// TwinCAT 3 PLC project FactoryIOPLCProject
// ProgramVersion: 3.1.4026.24
// libraries:
//   Tc2_ModbusSrv, * (Beckhoff Automation GmbH)
//   Tc2_Standard, * (Beckhoff Automation GmbH)
//   Tc2_System, * (Beckhoff Automation GmbH)
//   Tc2_Utilities, * (Beckhoff Automation GmbH)
// project tree:
//   DUTs/Communication/ADS/ ADSCommunicationInterface.TcDUT (not stored)
//   DUTs/HMI/Header/ HMIHeader.TcDUT
//   DUTs/HMI/MachineSection/ HMIMovementForkInterface.TcDUT, HMIMovementInterface.TcDUT, HMIRFIDControlInterface.TcDUT (not stored), HMIRFIDDataInterface.TcDUT (not stored), HMIRFIDInterface.TcDUT, HMIRFIDStatusInterface.TcDUT, HMIRuncontrolInterface.TcDUT, HMIWindowSwitch.TcDUT, HMIWorkpieceInterface.TcDUT, MachineSection.TcDUT, MachineSectionHMIInterface.TcDUT
//   DUTs/HMI/NumericalInput/ HMIButtonNumericalInputInterface.TcDUT, HMINumericalInputInterface.TcDUT (not stored), HMINumericalInputLineInterface.TcDUT
//   DUTs/HMI/SettingLine/ HMIButtonSettingLineInterface.TcDUT, HMISettingLineInterface.TcDUT
//   DUTs/OperatingMode/ ActionState.TcDUT, FaultWarningState.TcDUT (not stored), HMIActionState.TcDUT, HMIInterfaceOperatingMode.TcDUT (not stored), HMIToPLCOperatingMode.TcDUT, OperatingMode.TcDUT (not stored), OperatingModeHomeing.TcDUT, PLCToHMIOperatingMode.TcDUT
//   DUTs/PickPlace/ PickPlacePosition.TcDUT
//   DUTs/PositingBar/ PositingBarAlignmentDirection.TcDUT (not stored)
//   DUTs/Program/PickPlace/ PickPlaceSteps.TcDUT
//   DUTs/Program/Warehouse/ StackerCraneSteps.TcDUT (not stored)
//   DUTs/RFID/ RFIDReadSerialnumberStates.TcDUT, RFIDReadWriteDataStates.TcDUT (not stored)
//   DUTs/VisionSensor/ VisionSensorParttype.TcDUT (not stored)
//   GVLs/ ADS_Communication.TcGVL, Elevator.TcGVL, Emitter.TcGVL, Foerderband.TcGVL, GVL.TcGVL, HMI.TcGVL, PickPlace.TcGVL, PositioningBar.TcGVL, Remover.TcGVL, RFID.TcGVL, VisionSensor.TcGVL, Warehouse.TcGVL, _OperatingMode.TcGVL, _IO.TcGVL
//   / PlcTask.TcTTO (not stored)
//   POUs/Programm/ADS/ Call_ADSCommunication.TcPOU
//   POUs/Programm/Aufzug/ Call_Aufzug.TcPOU
//   POUs/Programm/Emitter/ Call_Emitter.TcPOU
//   POUs/Programm/Foerderband/ Call_Foerderband.TcPOU
//   POUs/Programm/HMI/ Call_HMI.TcPOU
//   POUs/Programm/ MAIN.TcPOU, SignalmappingInput.TcPOU, SignalmappingOutput.TcPOU
//   POUs/Programm/OperatingMode/ Call_OperatingMode.TcPOU
//   POUs/Programm/PickPlace/ Call_PickPlace.TcPOU
//   POUs/Programm/PositingBar/ Call_PositingBar.TcPOU
//   POUs/Programm/Remover/ Call_Remover.TcPOU
//   POUs/Programm/RFID/ Call_RFID.TcPOU
//   POUs/Programm/VisionSensor/ Call_VisionSensor.TcPOU
//   POUs/Programm/Warehouse/ Call_Warehouse.TcPOU
//   POUs/Vorlagen/AnalogValueHandling/ FC_AnalogInputValueHandling.TcPOU, FC_AnalogOutputValueHandling.TcPOU (not stored)
//   POUs/Vorlagen/Aufzug/ FB_Elevator.TcPOU
//   POUs/Vorlagen/Communication/ADS/ FB_ADSCommunicationStatus.TcPOU
//   POUs/Vorlagen/Emitter/ FB_Emitter.TcPOU
//   POUs/Vorlagen/Foerderband/ FB_Foerderband.TcPOU
//   POUs/Vorlagen/HMI/ FB_HMIHeader.TcPOU, FC_InitializingSettingLines.TcPOU
//   POUs/Vorlagen/OperatingMode/ FB_OperatingMode.TcPOU
//   POUs/Vorlagen/PickPlace/ FB_PickPlace_DigitalAnalog.TcPOU
//   POUs/Vorlagen/PositingBar/ FB_PositingBar.TcPOU
//   POUs/Vorlagen/Remover/ FB_Remover.TcPOU
//   POUs/Vorlagen/RFID/ FB_RFID.TcPOU
//   POUs/Vorlagen/VisionSensor/ FB_VisionSensor.TcPOU
//   POUs/Vorlagen/Warehouse/ FB_StackerCrane_Analog.TcPOU (not stored), FB_StackerCrane_Numerical.TcPOU
// real-time tasks:
//   TASK PlcTask: cycle T#10ms, priority 20, ADS port 350

// ---- DUTs/HMI/Header/HMIHeader.TcDUT
TYPE HMIHeader :
STRUCT
	PathOperatingMode	:	STRING;
	PathMachineState	:	STRING;
	NameApplication	:	STRING;
	ErrorIsActive	:	BOOL;
	State	:	INT;
END_STRUCT
END_TYPE

// ---- DUTs/HMI/MachineSection/HMIMovementForkInterface.TcDUT
TYPE HMIMovementForkInterface :
STRUCT
	ForkMovementButtons	:	ARRAY [1..8] of HMIButtonMachineSection;
END_STRUCT
END_TYPE

// ---- DUTs/HMI/MachineSection/HMIMovementInterface.TcDUT
TYPE HMIMovementInterface :
STRUCT
	MovementSettingLines	:	ARRAY [1..3] of HMISettingLineInterface;
END_STRUCT
END_TYPE

// ---- DUTs/HMI/MachineSection/HMIRFIDInterface.TcDUT
TYPE HMIRFIDInterface :
STRUCT
	PermissionHardware	:	BOOL;
	PartPresent	:	BOOL;
	ExecuteCommand	:	BOOL;
	FMReading	:	BOOL;
	FMWritting	:	BOOL;
	ErrorActive	:	BOOL;
	SelectedCommand	:	WORD;
	ReadValue	:	WORD;
	WriteValue	:	WORD;
	SelectedMemoryIndex	:	WORD;
	StatusReader	:	WORD;
	CommandID	:	WORD;
	AllReadData	:	ARRAY[0..127] OF WORD;
	AllWriteData	:	ARRAY[0..127] OF WORD;
END_STRUCT
END_TYPE

// ---- DUTs/HMI/MachineSection/HMIRFIDStatusInterface.TcDUT
TYPE HMIRFIDStatusInterface :
STRUCT
	PermissionHardware	:	BOOL;
	PartPresent	:	BOOL;
	ErrorActive	:	BOOL;
	FMReading	:	BOOL;
	FMWritting	:	BOOL;
END_STRUCT
END_TYPE

// ---- DUTs/HMI/MachineSection/HMIRuncontrolInterface.TcDUT
TYPE HMIRuncontrolInterface :
STRUCT
	RuncontrolButtons	:	ARRAY [1..10] of HMIButtonMachineSection;
END_STRUCT
END_TYPE

// ---- DUTs/HMI/MachineSection/HMIWindowSwitch.TcDUT
TYPE HMIWindowSwitch :
STRUCT
	MinPage	:	INT;
	MaxPage	:	INT;
	SelectedPage	:	INT;
	SelectedTab	:	STRING;
	NextPageIsEnabled	:	BOOL;
	NextPageIsPressed	:	BOOL;
	PreviousPageIsEnabled	:	BOOL;
	PreviousPageIsPressed	:	BOOL;
END_STRUCT
END_TYPE

// ---- DUTs/HMI/MachineSection/HMIWorkpieceInterface.TcDUT
TYPE HMIWorkpieceInterface :
STRUCT
	WorkpieceSettingLines	:	ARRAY[1..3] of HMISettingLineInterface;	
END_STRUCT
END_TYPE

// ---- DUTs/HMI/MachineSection/MachineSection.TcDUT
{attribute 'qualified_only'}
{attribute 'strict'}
{attribute 'to_string'}
TYPE MachineSection :
(
	None := 0,
	Conveyor,
	Emitter,
	Elevator,
	StackerCrane,
	RFID,
	PositingBar,
	PickPlace,
	Remover
);
END_TYPE

// ---- DUTs/HMI/MachineSection/MachineSectionHMIInterface.TcDUT
TYPE MachineSectionHMIInterface :
STRUCT
	ActiveMachineSection : MachineSection;
	SelectedActor : INT;
	PageSwitch	:	HMIWindowSwitch;
	Movements : HMIMovementInterface;
	Forks : HMIMovementForkInterface;
	Runcontrols : HMIRuncontrolInterface;
	RFID : HMIRFIDInterface;
	Workpiece : HMIWorkpieceInterface;
END_STRUCT
END_TYPE

// ---- DUTs/HMI/NumericalInput/HMIButtonNumericalInputInterface.TcDUT
TYPE HMIButtonNumericalInputInterface :
STRUCT
	IsEnabled	:	BOOL;
	IsPressed	:	BOOL;
	InPosition	:	BOOL;
	IsVisibleButton	:	BOOL;
	CaptionButton	:	STRING;
	PathImageButton	:	STRING;
END_STRUCT
END_TYPE

// ---- DUTs/HMI/NumericalInput/HMINumericalInputLineInterface.TcDUT
TYPE HMINumericalInputLineInterface :
STRUCT
	CaptionDescription	:	STRING;
	UnitInput	:	STRING;
	ValueInput	:	REAL;
	IsEnabledInput	:	BOOL;
END_STRUCT
END_TYPE

// ---- DUTs/HMI/SettingLine/HMIButtonSettingLineInterface.TcDUT
TYPE HMIButtonSettingLineInterface :
STRUCT
	IsEnabled	:	BOOL;
	IsPressed	:	BOOL;
	InPosition	:	BOOL;
	IsVisibleAxisPosition	:	BOOL;
	IsVisibleButton	:	BOOL;
	AxisPosition	:	REAL;
	CaptionButton	:	STRING;
	PathImageButton	:	STRING;
END_STRUCT
END_TYPE

// ---- DUTs/HMI/SettingLine/HMISettingLineInterface.TcDUT
TYPE HMISettingLineInterface :
STRUCT
	CaptionSettingLine	:	STRING;
	VisibilitySettingLine	:	BOOL;
	SettingLineButtons	:	ARRAY[1..3] OF HMIButtonSettingLineInterface;
END_STRUCT
END_TYPE

// ---- DUTs/OperatingMode/ActionState.TcDUT
TYPE ActionState :
STRUCT
	PreconditionsFullfilled	:	BOOL;
	IsActive	:	BOOL;
END_STRUCT
END_TYPE

// ---- DUTs/OperatingMode/HMIActionState.TcDUT
TYPE HMIActionState :
STRUCT
	IsSelected	:	BOOL;
END_STRUCT
END_TYPE

// ---- DUTs/OperatingMode/HMIToPLCOperatingMode.TcDUT
TYPE HMIToPLCOperatingMode :
STRUCT
	Manuel	:	HMIActionState;
	Automatic	:	HMIActionState;
	AutomaticStart	:	HMIActionState;
	AutomaticStop	:	HMIActionState;
	Quit	:	HMIActionState;
	Reset	:	HMIActionState;
END_STRUCT
END_TYPE

// ---- DUTs/OperatingMode/OperatingModeHomeing.TcDUT
TYPE OperatingModeHomeing :
STRUCT
	PreconditionsFullfilled	:	BOOL;
	IsActive	:	BOOL;
	IsReached	:	BOOL;
	AllMachinesInHome	:	BOOL;
END_STRUCT
END_TYPE

// ---- DUTs/OperatingMode/PLCToHMIOperatingMode.TcDUT
TYPE PLCToHMIOperatingMode :
STRUCT
	CurrentOperatingMode	:	OperatingMode;	
END_STRUCT
END_TYPE

// ---- DUTs/PickPlace/PickPlacePosition.TcDUT
TYPE PickPlacePosition :
STRUCT
	PositionXAxis	:	REAL;
	PositionYAxis	:	REAL;
	PositionZAxis	:	REAL;
	PositionCAxis	:	REAL;
END_STRUCT
END_TYPE

// ---- DUTs/Program/PickPlace/PickPlaceSteps.TcDUT
{attribute 'qualified_only'}
{attribute 'strict'}
{attribute 'to_string'}
TYPE PickPlaceSteps :
(
	WaitingForAutomaticStart := 0,
	DriveToHome,
	DriveXYToPick,
	DriveZDown,
	GrabPart,
	DriveZUp
);
END_TYPE

// ---- DUTs/RFID/RFIDReadSerialnumberStates.TcDUT
{attribute 'qualified_only'}
{attribute 'strict'}
{attribute 'to_string'}
TYPE RFIDReadSerialnumberStates :
(
	WAITINGTRIGGER := 0,
	SETTRIGGER,
	WAITINGRESPONSE,
	RESPONSE,
	ERRORACTIVE
);
END_TYPE

// ---- GVLs/ADS_Communication.TcGVL
VAR_GLOBAL
	Data_Ready	:	BOOL;
	Detected_Material	:	INT;
	
	RF_Data_Ready	:	R_TRIG;
END_VAR

// ---- GVLs/Elevator.TcGVL
VAR_GLOBAL
	AufzugSensorEinlaufFoerderband	:	BOOL;
	AufzugSensorAuslaufFoerderband	:	BOOL;
	AufzugFoerderbandVorwaerts	:	BOOL;
	AufzugFoerderbandRueckwaerts	:	BOOL;
	AufzugSollwert	:	WORD;
	AufzugIstwert	:	WORD;
	
	(*======================= Simulation* =======================*)
	IstPositionConverted	:	REAL;
	SollPosition	:	REAL;
	AufzugInPosition	:	BOOL;
	AufzugBewegen	:	BOOL;
	AufzugFoerderbandVor	: BOOL;
	AufzugFoerderbandRueck	: BOOL;
	AufzugFoerderbandStop	: BOOL;
	instFBElevator	:	FB_Elevator;
END_VAR

// ---- GVLs/Emitter.TcGVL
VAR_GLOBAL
	instEmitter	:	FB_Emitter;	//Instanz Emitter 4m Rollenfoerderer
	CreateNewPart	:	BOOL;
END_VAR

// ---- GVLs/Foerderband.TcGVL
VAR_GLOBAL
	Sensor_Band_Einlauf	:	BOOL;	//Sensor am Band Anfang
	Sensor_Band_Auslauf	:	BOOL;	//Sensor am Band Ende
	Foerderband_Vorwaerts	:	BOOL;	//Foerdreband Motor vorwaerts drehen
	Foerderband_Rueckwaerts	:	BOOL;	//Foerderband Motor ruechwaerts drehen
	
	(* ==================================== Simulation signals ====================================*)
	instFoerderband6	:	FB_Foerderband;
END_VAR

// ---- GVLs/GVL.TcGVL
{attribute 'qualified_only'}
VAR_GLOBAL
	//Hier die Array-Grenzen anpassen auf die maximale Anzahl an Signalen.
	//Der Name der Liste, darf nicht verändert werden.
	mb_Input_Coils        : ARRAY [0..255] OF BOOL;	//Digital outputs of the PLC
    mb_Output_Coils       : ARRAY [0..255] OF BOOL;	//Digital inputs of the PLC
    mb_Input_Registers    : ARRAY [0..255] OF WORD;	//Analog outputs of the PLC
    mb_Output_Registers   : ARRAY [0..255] OF WORD;	//Analog inputs of the PLC	
END_VAR

// ---- GVLs/HMI.TcGVL
VAR_GLOBAL
	hmiHeaderInstance	:	FB_HMIHeader;
	hmiHeaderInterface	:	HMIHeader;	
	hmiOperatingmodeInterface	:	HMIInterfaceOperatingMode;
	
	hmiAdsCommunicationInterfaceInstance	:	FB_ADSCommunicationStatus;
	hmiAdsCommunicationInterface	:	ADSCommunicationInterface;
	
	hmiMachineSectionInterface	:	MachineSectionHMIInterface;
	
	hmiEmitterInstances	:	ARRAY[0..1] OF STRING := [
														'Zufuehrband',
														'SubParts'
													];
	hmiConveyorInstances	:	ARRAY[0..1] OF STRING := [
															'Foerderband 6',
															'Zufuehrung'
														 ];
	hmiElevatorInstances	:	ARRAY[0..1] OF STRING := [
															'Einlauf',
															'Hochregallager'
														];
	hmiStackerCraneInstances	:	ARRAY[0..1] OF STRING := [
															'Einlagerung',
															'Auslagerung'
														 ];		
	hmiRFIDInstances	:	ARRAY[0..2] OF STRING := [
															'Einlagerung',
															'Zufuehrung',
															'Warehouse-Infeed'
														 ];	
	hmiPositingBarInstances	:	ARRAY[0..2] OF STRING := [
															'Blau laden',
															'Gruen laden',
															'Grau laden'
														 ];										 
	hmiPickPlaceInstances	:	ARRAY[0..2] OF STRING := [
															'Einlagerung',
															'Zufuehrung',
															'Warehouse-Infeed'
														 ];	
	hmiRemoverInstances	:	ARRAY[0..1] OF STRING := [
														'Zufuehrband',
														'SubParts'
													];
END_VAR

// ---- GVLs/PickPlace.TcGVL
VAR_GLOBAL
	PickPlaceBoxDetected	:	BOOL;
	PickPlaceCAxisInPos	:	BOOL;
	PickPlaceZAxisIsMoving	:	BOOL;
	PickPlaceX_YAxisIsMoving	:	BOOL;
	
	PickPlaceCAxisMovePlus	:	BOOL;
	PickPlaceGrabBox	:	BOOL;
	
	PickPlacePositionYAxis	:	WORD;
	PickPlacePositionZAxis	:	WORD;
	PickPlacePositionXAxis	:	WORD;
	
	PickPlaceSetpositionYAxis	:	WORD;
	PickPlaceSetpositionZAxis	:	WORD;
	PickPlaceSetpositionXAxis	:	WORD;
	
	(*========================== Simulation ==========================*)
	instPickPlaceDigitalAnalog	:	FB_PickPlace_DigitalAnalog;
	processStepsPickPlace	:	PickPlaceSteps;
	HomePosition	:	PickPlacePosition{
						PositionXAxis := 0.0,
						PositionYAxis := 0.0,
						PositionZAxis := 0.0,
						PositionCAxis := 0.0
						};
	PickPlacePosition	:	PickPlacePosition{
						PositionXAxis := 1.0,
						PositionYAxis := 1.0,
						PositionZAxis := 1.0,
						PositionCAxis := 0.0
						};
	WaitingTimeGrabPart	:	TON;
	
	DelayProcessStep	:	BOOL;
END_VAR

// ---- GVLs/PositioningBar.TcGVL
VAR_GLOBAL
	PositionerIsClamped	:	BOOL;
	PositionerIsRaised	:	BOOL;
	PositionerClamp	:	BOOL;
	PositionerRaise	:	BOOL;
	instControlBlockPositingBar	:	FB_PositingBar;
	
	(*================== Simulation ==================*)
	SimuClampPositingBar	:	BOOL;
	SimuUnclampPositingBar	:	BOOL;
	SimuRaisePositingBar	:	BOOL;
	SimuLowerPositingBar	:	BOOL;
END_VAR

// ---- GVLs/Remover.TcGVL
VAR_GLOBAL
	RemoverPartPresent	:	BOOL;
	Remover	:	BOOL;
	
	(*=================== Simu ===================*)
	instFBRemover	:	FB_Remover;
	
END_VAR

// ---- GVLs/RFID.TcGVL
VAR_GLOBAL
	RFIDCommandID	:	WORD;
	RFIDReadData	:	WORD;
	RFIDStatus	:	WORD;
	RFIDExecuteCommand	:	BOOL;
	RFIDCommand	:	WORD;
	RFIDWriteData	:	WORD;
	RFIDMemoryIndex	:	WORD;
	(*======================== Simulation ========================*)
	RFIDReadSerialNumberSimu	:	BOOL;
	RFIDReadDataSimu	:	BOOL;
	RFIDWriteDataSimu	:	BOOL;
	RFIDCompleteDataToReadSimu	:	ARRAY[0..127] of WORD;
	RFIDCompleteDataToWriteSimu	:	ARRAY[0..127] of WORD;
	instFBRFID	:	FB_RFID;
END_VAR

// ---- GVLs/VisionSensor.TcGVL
VAR_GLOBAL
	PartDetectedVisionSensor	:	BOOL;
	ErrorVisionSensor	:	BOOL;
	ReadPartCode	:	WORD;
	
	instVisionSensorConveyor	:	FB_VisionSensor;
END_VAR

// ---- GVLs/Warehouse.TcGVL
VAR_GLOBAL
	(*======================= Analog Stacker crane* =======================*)
	RBGEndlageMitte	:	BOOL;
	RBGEndlageLinks	:	BOOL;
	RBGEndlageRechts :	BOOL;
	RBGIstwertX	:	WORD;
	RBGIstwertZ	:	WORD;
	RBGGabelLinks	:	BOOL;
	RBGGabelRechts	:	BOOL;
	RBGSollwertX	:	WORD;
	RBGSollwertZ	:	WORD;
	
(*======================= Simulation* =======================*)
	RBGStartMove	:	BOOL;
	RBGStartForkLeftMove	:	BOOL;
	RBGStartForkRightMove	:	BOOL;
	RBGStartForkMiddleMove	:	BOOL;
	InUnloadingAnalog	:	BOOL;
	RBGSollwertXSimu	:	REAL;
	RBGSollwertZSimu	:	REAL;
	instStackerCraneAnalog	:	FB_StackerCrane_Analog;
	processStepsAnalogStackerCrane	: StackerCraneSteps;
	
(*======================= Numerical Stacker crane* =======================*)	
	DigitalStackerCraneEndlageMitte	:	BOOL;
	DigitalStackerCraneEndlageLinks	:	BOOL;
	DigitalStackerCraneEndlageRechts :	BOOL;
	DigitalStackerCraneGabelLinks	:	BOOL;
	DigitalStackerCraneGabelRechts	:	BOOL;
	DigitalStackerCraneLiftGabel	:	BOOL;
	DigitalStackerCraneXAxisIsMoving	:	BOOL;
	DigitalStackerCraneZAxisIsMoving	:	BOOL;
	DigitalStackerCraneTargetPos	:	WORD;
	
	(*======================= Simulation* =======================*)
	DigtalStackerCraneStartMove	:	BOOL;
	DigtalStackerCraneStartForkLeftMove	:	BOOL;
	DigtalStackerCraneStartForkRightMove	:	BOOL;
	DigtalStackerCraneStartForkMiddleMove	:	BOOL;
	DigitalStackerCraneStartLiftFork	:	BOOL;
	InUnloadingNumerical	:	BOOL;
	Lifting	:	BOOL;
	Lowering	:	BOOL;
	DigitalTargetPosSimu	:	WORD := 7;
	instStackerCraneNumerical	:	FB_StackerCrane_Numerical;
	processStepsNumericalStackerCrane	: StackerCraneSteps;
END_VAR

// ---- GVLs/_OperatingMode.TcGVL
VAR_GLOBAL
	(* ==================================== Buttons ====================================*)
	BetrMan		:	BOOL;	//Betriebsart Manuell
	BetrAuto	:	BOOL;	//Betriebsart Auto
	StartButton	:	BOOL;	//Start-Button
	StopButton	:	BOOL;	//Stop-Button
	HomeButton	:	BOOL;	//Grundstellungsbutton
	ResetButton	:	BOOL;	//Reset-Button
	QuitButton	:	BOOL;	//Quit-Button
	E_Stop		:	BOOL;	//Not-Aus
	(* ==================================== LED's ====================================*)
	StartLED	:	BOOL;	//LED-Start
	StopLED		:	BOOL;	//LED-Stop
	HomeLED		:	BOOL;	//LED-Grundstellung
	ResetLED	:	BOOL;	//LED-Reset
	QuitLED		:	BOOL;	//LED-Quit
	
	(* ==================================== Simulation signals ====================================*)
	instOperatingMode	:	FB_OperatingMode;
	simPermissionHardware	:	BOOL;
	simPermissionSafety		:	BOOL;
END_VAR

// ---- GVLs/_IO.TcGVL
VAR_GLOBAL
	
	(* ==================================== Digitale Eingaenge ====================================*)
	
	BauteilVorEmitter	:	BOOL;	//Sensor 4m Rollenband Emitter Bauteil vorhanden
	(* ==================================== Digitale Ausgaenge ====================================*)
	
	Emitter_Rollenband4m	:	BOOL;	//Emitter Rollenband 4m hinten im Eck
END_VAR

// ---- POUs/Vorlagen/Aufzug/FB_Elevator.TcPOU
FUNCTION_BLOCK FB_Elevator
VAR_INPUT
	CurrentPosition	:	WORD;	//Current Position of Conveyor
	SensorOutfeed	:	BOOL;	//Sensor Outfeed Conveyor
	SensorInfeed	:	BOOL;	//Sensor Infeed Conveyor
	ActorInstanceIndex	:	INT;	//Index in DropDown HMI
	ActorInstanceName	:	STRING;		//Name of the instance
END_VAR
VAR_OUTPUT
	SetPointPositionElevator	:	WORD;
	ConveyorForward		:	BOOL;
	ConveyorBackward	:	BOOL;
	ElevatorInPosition	:	BOOL;
END_VAR
VAR_IN_OUT
	OperatingMode	:	OperatingMode;	//Schnittstelle für Betriebsarten
	HMIInterface	:	MachineSectionHMIInterface;	//HMI-Interface
END_VAR
VAR
	statCurrentPosition	:	REAL;
	statSetPointPosition	:	REAL;	
	statSelectedPositionToElevator	:	REAL;
	statPositionToElevator	:	WORD;
	statConveyorForward		:	BOOL;
	statConveyorBackward	:	BOOL;
	statMoveElevator	:	BOOL;
	statInPosition	:	BOOL;
	statRTrigPartOutfeed	:	R_TRIG;
	statRTrigPartInfeed	:	R_TRIG;
	
	internHMIInterface	:	MachineSectionHMIInterface;
	internInstanceActivatedFirstTime	:	BOOL;
	internRisingEdgePressButtonUpElevator	:	R_TRIG;
	internRisingEdgePressButtonDownElevator	:	R_TRIG;
	internRisingEdgePressButtonStopElevator	:	R_TRIG;
	internRisingEdgePressButtonForwardConveyor	:	R_TRIG;
	internRisingEdgePressButtonBackwardConveyor	:	R_TRIG;
	internRisingEdgePressButtonStopConveyor	:	R_TRIG;
	internStopElevator	:	BOOL;
	internStopConveyor	:	BOOL;
	internUpMovingElevator	:	BOOL;
	internDownMovingElevator	:	BOOL;
END_VAR

(*===================== CurrentPosition =====================*)
FC_AnalogInputValueHandling(RowValue:= CurrentPosition, 
							UpperLimit:= 7.0, 
							LowerLimit:= 0.0, 
							ConvertedValue=> statCurrentPosition);
							
(*===================== HMI INTERFACE =====================*)
internHMIInterface := HMIInterface;

IF internHMIInterface.ActiveMachineSection = MachineSection.Elevator AND
	internHMIInterface.SelectedActor = ActorInstanceIndex THEN
	(*===================== Initializing HMI-Interface =====================*)
	IF NOT internInstanceActivatedFirstTime THEN
		FC_InitializingSettingLines(HMIInterface := internHMIInterface);
		internInstanceActivatedFirstTime := TRUE;
	END_IF
	(*===================== Button Handling Movement =====================*)
	internHMIInterface.Movements.MovementSettingLines[1].CaptionSettingLine := CONCAT('Elevator Axis Control ', ActorInstanceName);
	internHMIInterface.Movements.MovementSettingLines[1].VisibilitySettingLine := TRUE;
	
	internHMIInterface.Movements.MovementSettingLines[1].SettingLineButtons[1].IsVisibleButton := TRUE;
	internHMIInterface.Movements.MovementSettingLines[1].SettingLineButtons[1].IsVisibleAxisPosition := FALSE;
	internHMIInterface.Movements.MovementSettingLines[1].SettingLineButtons[1].IsEnabled := OperatingMode.ManuelIsActive AND NOT
									 														OperatingMode.EStop.IsActive AND NOT
																							OperatingMode.Fault.IsActive AND NOT
																							statMoveElevator AND
																							statSetPointPosition < 7;
	internHMIInterface.Movements.MovementSettingLines[1].SettingLineButtons[1].InPosition := internUpMovingElevator;
	internHMIInterface.Movements.MovementSettingLines[1].SettingLineButtons[1].CaptionButton := 'Up';
	internHMIInterface.Movements.MovementSettingLines[1].SettingLineButtons[1].PathImageButton := 'Images\UpElevator.svg';
	
	internHMIInterface.Movements.MovementSettingLines[1].SettingLineButtons[2].IsVisibleButton := TRUE;
	internHMIInterface.Movements.MovementSettingLines[1].SettingLineButtons[2].IsVisibleAxisPosition := TRUE;
	internHMIInterface.Movements.MovementSettingLines[1].SettingLineButtons[2].IsEnabled := OperatingMode.ManuelIsActive;
	internHMIInterface.Movements.MovementSettingLines[1].SettingLineButtons[2].InPosition := NOT statMoveElevator;
	internHMIInterface.Movements.MovementSettingLines[1].SettingLineButtons[2].AxisPosition := statCurrentPosition;
	internHMIInterface.Movements.MovementSettingLines[1].SettingLineButtons[2].CaptionButton := 'Stop';
	internHMIInterface.Movements.MovementSettingLines[1].SettingLineButtons[2].PathImageButton := 'Images\StopConveyor.svg';
	
	internHMIInterface.Movements.MovementSettingLines[1].SettingLineButtons[3].IsVisibleButton := TRUE;
	internHMIInterface.Movements.MovementSettingLines[1].SettingLineButtons[3].IsVisibleAxisPosition := FALSE;
	internHMIInterface.Movements.MovementSettingLines[1].SettingLineButtons[3].IsEnabled := OperatingMode.ManuelIsActive AND NOT
									 														OperatingMode.EStop.IsActive AND NOT
																							OperatingMode.Fault.IsActive AND NOT
																							statMoveElevator AND
																							statSetPointPosition > 0;
	internHMIInterface.Movements.MovementSettingLines[1].SettingLineButtons[3].InPosition := internDownMovingElevator;
	internHMIInterface.Movements.MovementSettingLines[1].SettingLineButtons[3].CaptionButton := 'Down';
	internHMIInterface.Movements.MovementSettingLines[1].SettingLineButtons[3].PathImageButton := 'Images\DownElevator.svg';
	
	internHMIInterface.Movements.MovementSettingLines[2].CaptionSettingLine := CONCAT('Elevator Conveyor Control ', ActorInstanceName);
	internHMIInterface.Movements.MovementSettingLines[2].VisibilitySettingLine := TRUE;
	
	internHMIInterface.Movements.MovementSettingLines[2].SettingLineButtons[1].IsVisibleButton := TRUE;
	internHMIInterface.Movements.MovementSettingLines[2].SettingLineButtons[1].IsVisibleAxisPosition := FALSE;
	internHMIInterface.Movements.MovementSettingLines[2].SettingLineButtons[1].IsEnabled := OperatingMode.ManuelIsActive AND NOT
									 														OperatingMode.EStop.IsActive AND NOT
																							OperatingMode.Fault.IsActive AND NOT
																							statMoveElevator AND NOT
																							statConveyorBackward AND
																							statInPosition;
	internHMIInterface.Movements.MovementSettingLines[2].SettingLineButtons[1].InPosition := statMoveElevator;
	internHMIInterface.Movements.MovementSettingLines[2].SettingLineButtons[1].CaptionButton := 'Forward';
	internHMIInterface.Movements.MovementSettingLines[2].SettingLineButtons[1].PathImageButton := 'Images\ForwardConveyor.svg';
	
	internHMIInterface.Movements.MovementSettingLines[2].SettingLineButtons[2].IsVisibleButton := TRUE;
	internHMIInterface.Movements.MovementSettingLines[2].SettingLineButtons[2].IsVisibleAxisPosition := FALSE;
	internHMIInterface.Movements.MovementSettingLines[2].SettingLineButtons[2].IsEnabled := OperatingMode.ManuelIsActive;
	internHMIInterface.Movements.MovementSettingLines[2].SettingLineButtons[2].InPosition := NOT statMoveElevator;
	internHMIInterface.Movements.MovementSettingLines[2].SettingLineButtons[2].CaptionButton := 'Stop';
	internHMIInterface.Movements.MovementSettingLines[2].SettingLineButtons[2].PathImageButton := 'Images\StopConveyor.svg';
	
	internHMIInterface.Movements.MovementSettingLines[2].SettingLineButtons[3].IsVisibleButton := TRUE;
	internHMIInterface.Movements.MovementSettingLines[2].SettingLineButtons[3].IsVisibleAxisPosition := FALSE;
	internHMIInterface.Movements.MovementSettingLines[2].SettingLineButtons[3].IsEnabled := OperatingMode.ManuelIsActive AND NOT
									 														OperatingMode.EStop.IsActive AND NOT
																							OperatingMode.Fault.IsActive AND NOT
																							statMoveElevator AND NOT
																							statConveyorBackward AND
																							statInPosition;
	internHMIInterface.Movements.MovementSettingLines[2].SettingLineButtons[3].InPosition := statMoveElevator;
	internHMIInterface.Movements.MovementSettingLines[2].SettingLineButtons[3].CaptionButton := 'Backward';
	internHMIInterface.Movements.MovementSettingLines[2].SettingLineButtons[3].PathImageButton := 'Images\BackwardConveyor.svg';
	
	(*===================== Elevator Up =====================*)
	internRisingEdgePressButtonUpElevator(CLK := internHMIInterface.Movements.MovementSettingLines[1].SettingLineButtons[1].IsPressed);
	IF internRisingEdgePressButtonUpElevator.Q THEN
		statSetPointPosition := statSetPointPosition + 0.2;
		statMoveElevator := TRUE;
		internUpMovingElevator := TRUE;
	END_IF
	(*===================== Elevator Down =====================*)
	internRisingEdgePressButtonDownElevator(CLK := internHMIInterface.Movements.MovementSettingLines[1].SettingLineButtons[3].IsPressed);
	IF internRisingEdgePressButtonDownElevator.Q THEN
		statSetPointPosition := statSetPointPosition - 0.2;
		statMoveElevator := TRUE;
		internDownMovingElevator := TRUE;
	END_IF
	(*===================== Elevator Stop =====================*)
	internRisingEdgePressButtonStopElevator(CLK := internHMIInterface.Movements.MovementSettingLines[1].SettingLineButtons[2].IsPressed);
	IF internRisingEdgePressButtonStopElevator.Q THEN
		internStopElevator := TRUE;
	END_IF
	(*===================== Conveyor Forward =====================*)
	internRisingEdgePressButtonForwardConveyor(CLK := internHMIInterface.Movements.MovementSettingLines[2].SettingLineButtons[1].IsPressed);
	IF internRisingEdgePressButtonForwardConveyor.Q THEN
		statConveyorForward := TRUE;
	END_IF
	(*===================== Conveyor Backward =====================*)
	internRisingEdgePressButtonBackwardConveyor(CLK := internHMIInterface.Movements.MovementSettingLines[2].SettingLineButtons[3].IsPressed);
	IF internRisingEdgePressButtonBackwardConveyor.Q THEN
		statConveyorBackward := TRUE;
	END_IF
	(*===================== Conveyor Stop =====================*)
	internRisingEdgePressButtonStopConveyor(CLK := internHMIInterface.Movements.MovementSettingLines[2].SettingLineButtons[2].IsPressed);
	IF internRisingEdgePressButtonStopConveyor.Q THEN
		internStopConveyor := TRUE;
	END_IF
	
	(*===================== Write Interface =====================*)
	HMIInterface := internHMIInterface;
ELSE
		internInstanceActivatedFirstTime := FALSE;
END_IF

(*===================== Elevator in Position =====================*)
IF (statCurrentPosition >= statSetPointPosition - 0.1) AND (statCurrentPosition <= statSetPointPosition + 0.1) THEN
	statInPosition := TRUE;
	statMoveElevator := FALSE;
	internUpMovingElevator := FALSE;
	internDownMovingElevator := FALSE;
ELSE
	statInPosition := FALSE;
END_IF
(*===================== Positioning Elevator =====================*)
IF (OperatingMode.AutomaticIsActive AND OperatingMode.AutomaticStart.IsActive) OR
	OperatingMode.ManuelIsActive AND statMoveElevator 
THEN
	statSelectedPositionToElevator := statSetPointPosition;
END_IF
IF OperatingMode.EStop.IsActive OR OperatingMode.Fault.IsActive OR 
   (OperatingMode.AutomaticIsActive AND OperatingMode.AutomaticStop.IsActive) OR
   (OperatingMode.ManuelIsActive AND internStopElevator)
THEN
	statSelectedPositionToElevator := statCurrentPosition;
	statMoveElevator := FALSE;
	internStopElevator := FALSE;
	internUpMovingElevator := FALSE;
	internDownMovingElevator := FALSE;
END_IF
(*===================== SetPointPosition =====================*)
FC_AnalogOutputValueHandling(Setpoint:= statSelectedPositionToElevator, 
						     UpperLimit:= 7.0, 
							 LowerLimit:= 0.0, 
							 ConvertedValue=> statPositionToElevator);
(*===================== Conveyor Reset =====================*)
IF OperatingMode.EStop.IsActive OR OperatingMode.Fault.IsActive OR 
(OperatingMode.AutomaticIsActive AND OperatingMode.AutomaticStop.IsActive) OR
(OperatingMode.ManuelIsActive AND internStopConveyor) 
THEN
	statConveyorForward := FALSE;
	statConveyorBackward := FALSE;
	internStopConveyor := FALSE;
END_IF
(*===================== Conveyor Forward =====================*)
statRTrigPartOutfeed(CLK:= SensorOutfeed);
IF statRTrigPartOutfeed.Q THEN
	statConveyorForward := FALSE;
END_IF
(*===================== Conveyor Backward =====================*)
statRTrigPartInfeed(CLK:= SensorInfeed);
IF statRTrigPartInfeed.Q THEN
	statConveyorBackward := FALSE;
END_IF
(*===================== Outputs writting =====================*)
SetPointPositionElevator := statPositionToElevator;
ConveyorForward := statConveyorForward;
ConveyorBackward := statConveyorBackward;
ElevatorInPosition := statInPosition;

METHOD PUBLIC Conveyor_OFF : BOOL
VAR_INPUT
	ConveyorStop	:	BOOL;
END_VAR
IF ConveyorStop THEN
	statConveyorForward := FALSE;
	statConveyorBackward := FALSE;
	Conveyor_OFF := TRUE;
END_IF
END_METHOD

METHOD PUBLIC ConveyorBackward_ON : BOOL
VAR_INPUT
	ConveyorBackwardStart	:	BOOL;
END_VAR
IF OperatingMode.AutomaticIsActive AND OperatingMode.AutomaticStart.IsActive AND 
	statInPosition AND ConveyorBackwardStart AND NOT statConveyorForward
	THEN
	statConveyorBackward := TRUE;
	ConveyorBackward_ON := TRUE;
ELSE
	ConveyorBackward_ON := FALSE;
END_IF
END_METHOD

METHOD PUBLIC ConveyorForward_ON : BOOL
VAR_INPUT
	ConveyorForwardStart	:	BOOL;
END_VAR
IF OperatingMode.AutomaticIsActive AND OperatingMode.AutomaticStart.IsActive AND 
	statInPosition AND ConveyorForwardStart AND NOT statConveyorBackward
	THEN
	statConveyorForward := TRUE;
	ConveyorForward_ON := TRUE;
ELSE
	ConveyorForward_ON := FALSE;
END_IF
END_METHOD

METHOD PUBLIC MoveElevator
VAR_INPUT
	MoveStart	:	BOOL;
	NewPosition	:	REAL;
END_VAR
IF OperatingMode.AutomaticIsActive AND OperatingMode.AutomaticStart.IsActive AND MoveStart
	THEN
	statMoveElevator := TRUE;
	SetPointPosition := NewPosition;
END_IF
END_METHOD

PROPERTY PUBLIC SetPointPosition : REAL
GET
SetPointPosition := statSetPointPosition;
END_GET
SET
IF SetPointPosition <= 7.0 AND SetPointPosition >= 0.0 THEN
	statSetPointPosition := SetPointPosition;
END_IF
END_SET
END_PROPERTY

END_FUNCTION_BLOCK

// ---- POUs/Vorlagen/AnalogValueHandling/FC_AnalogInputValueHandling.TcPOU
FUNCTION FC_AnalogInputValueHandling
VAR_INPUT
	RowValue	:	WORD;	//Rohwert Sensor
	UpperLimit	:	REAL;	//Obere Grenze Umrechnungsbereich
	LowerLimit	:	REAL;	//Untere Grenze Umrechnungsbereich
END_VAR
VAR_OUTPUT
	ConvertedValue	:	REAL;	//Berechneter Wert
END_VAR
VAR
	tempConvertedRowValue	:	REAL;
	tempInputValueRange	:	REAL;
	tempCalculatedValue	:	REAL;
END_VAR

tempConvertedRowValue := TO_REAL(RowValue);
tempInputValueRange := tempConvertedRowValue / 100.0;
tempCalculatedValue := (tempInputValueRange * (UpperLimit - LowerLimit) / 10) + LowerLimit;

ConvertedValue := tempCalculatedValue;

END_FUNCTION

// ---- POUs/Vorlagen/HMI/FC_InitializingSettingLines.TcPOU
FUNCTION FC_InitializingSettingLines
VAR_IN_OUT
	HMIInterface	:	MachineSectionHMIInterface;
END_VAR
VAR
	internHMIInterface	:	MachineSectionHMIInterface;
	emptyHMIMovementInterface	:	HMIMovementInterface;
	emptyHMIMovementForkInterface	:	HMIMovementForkInterface;
	emptyHMIRuncontrolInterface	:	HMIRuncontrolInterface;
	emptyHMIRFIDInterface	:	HMIRFIDInterface;
	emptyHMIWorkpieceInterface	:	HMIWorkpieceInterface;
END_VAR

(*===================== Load Interface =====================*)
internHMIInterface := HMIInterface;

(*===================== Initializing Interface =====================*)
internHMIInterface.Movements := emptyHMIMovementInterface;
internHMIInterface.Forks := emptyHMIMovementForkInterface;
internHMIInterface.Runcontrols := emptyHMIRuncontrolInterface;
internHMIInterface.RFID := emptyHMIRFIDInterface;
internHMIInterface.Workpiece := emptyHMIWorkpieceInterface;
(*===================== Write Interface =====================*)
HMIInterface := internHMIInterface;

END_FUNCTION

// ---- POUs/Vorlagen/Emitter/FB_Emitter.TcPOU
FUNCTION_BLOCK FB_Emitter
VAR_INPUT
	PartPresent	:	BOOL;
	ActorInstanceIndex	:	INT;
	ActorInstanceName	:	STRING;
END_VAR
VAR_IN_OUT
	HMIInterface	:	MachineSectionHMIInterface;
END_VAR
VAR_OUTPUT
	CreatePart	:	BOOL;
END_VAR
VAR
	internCreatePart	: BOOL;
	
	internHMIInterface	:	MachineSectionHMIInterface;
	internInstanceActivatedFirstTime	:	BOOL;
	internRisingEdgePressButton	:	R_TRIG;
END_VAR

(*===================== HMI Interface =====================*)
internHMIInterface := HMIInterface;

IF internHMIInterface.ActiveMachineSection = MachineSection.Emitter AND
	internHMIInterface.SelectedActor = ActorInstanceIndex THEN
	(*===================== Initializing HMI-Interface =====================*)
	IF NOT internInstanceActivatedFirstTime THEN
		FC_InitializingSettingLines(HMIInterface := internHMIInterface);
		internInstanceActivatedFirstTime := TRUE;
	END_IF
	(*===================== Button Handling =====================*)
	internHMIInterface.Workpiece.WorkpieceSettingLines[1].CaptionSettingLine := CONCAT('Creation Part ', ActorInstanceName);
	internHMIInterface.Workpiece.WorkpieceSettingLines[1].VisibilitySettingLine := TRUE;
	
	internHMIInterface.Workpiece.WorkpieceSettingLines[1].SettingLineButtons[1].IsVisibleButton := TRUE;
	internHMIInterface.Workpiece.WorkpieceSettingLines[1].SettingLineButtons[1].IsVisibleAxisPosition := FALSE;
	internHMIInterface.Workpiece.WorkpieceSettingLines[1].SettingLineButtons[1].IsEnabled := NOT PartPresent;
	internHMIInterface.Workpiece.WorkpieceSettingLines[1].SettingLineButtons[1].InPosition := PartPresent;
	internHMIInterface.Workpiece.WorkpieceSettingLines[1].SettingLineButtons[1].CaptionButton := 'Create';
	internHMIInterface.Workpiece.WorkpieceSettingLines[1].SettingLineButtons[1].PathImageButton := 'Images\CreatePartEmitter.svg';
	
	internRisingEdgePressButton(CLK := internHMIInterface.Workpiece.WorkpieceSettingLines[1].SettingLineButtons[1].IsPressed);
	IF internRisingEdgePressButton.Q THEN
		internCreatePart := TRUE;
	END_IF
	(*===================== Write Interface =====================*)
	HMIInterface := internHMIInterface;
ELSE
		internInstanceActivatedFirstTime := FALSE;
END_IF
(*===================== Create Parts =====================*)
IF PartPresent THEN
	internCreatePart := FALSE;
END_IF

CreatePart := internCreatePart;

METHOD PUBLIC Create : BOOL
IF NOT PartPresent THEN
	internCreatePart := TRUE;
	Create := TRUE;
ELSE
	internCreatePart := FALSE;
	Create := FALSE;
END_IF
END_METHOD

END_FUNCTION_BLOCK

// ---- POUs/Vorlagen/Foerderband/FB_Foerderband.TcPOU
FUNCTION_BLOCK FB_Foerderband
VAR_INPUT
	SensorInfeed	:	BOOL;	//Sensor am Band Einlauf
	SensorOutfeed	:	BOOL;	//Sensor am Band Auslauf
	MaximumTimeRuncontrol	:	TIME;	//Maximale Zeit bis Fehler Laufkontrolle aktiviert wird
	ActorInstanceIndex	:	INT;
	ActorInstanceName	:	STRING;
END_VAR
VAR_IN_OUT
	HMIInterface	:	MachineSectionHMIInterface;
END_VAR
VAR_OUTPUT
	MotorForward	:	BOOL;	//Motor vorwaerts drehen
	MotorBackward	:	BOOL;	//Motor rueckwaerts drehen
	RuncontrolForwardActive	:	BOOL;	//Laufkontrolle in Vorwaerts-Richtung aktiv
	RuncontrolBackwardActive	:	BOOL;	//Laufkontrolle in Rueckwaerts-Richtung aktiv
	Error	:	BOOL;	//Fehler aktiv
END_VAR
VAR_IN_OUT
	OperatingMode	:	OperatingMode;	//Schnittstelle für Betriebsarten
END_VAR
VAR
	statMotorForward	:	BOOL;
	statMotorBackward	:	BOOL;
	statRuncontrolForward	:	BOOL;
	statRuncontrolBackward	:	BOOL;
	statErrorRuncontrolForward	:	BOOL;
	statErrorRuncontrolBackward	:	BOOL;
	statTimeRuncontrolForward	:	TON;
	statTimeRuncontrolBackward	:	TON;
	
	internHMIInterface	:	MachineSectionHMIInterface;
	internInstanceActivatedFirstTime	:	BOOL;
	internRisingEdgePressButtonForward	:	R_TRIG;
	internRisingEdgePressButtonBackward	:	R_TRIG;
	internRisingEdgePressButtonStop	:	R_TRIG;
	internRisingEdgePressButtonRuncontrolForwardReset	:	R_TRIG;
	internRisingEdgePressButtonRuncontrolBackwardReset	:	R_TRIG;
	internResetRuncontrolForward	:	BOOL;
	internResetRuncontrolBackward	:	BOOL;
END_VAR

(*===================== HMI INTERFACE =====================*)
internHMIInterface := HMIInterface;

IF internHMIInterface.ActiveMachineSection = MachineSection.Conveyor AND
	internHMIInterface.SelectedActor = ActorInstanceIndex THEN
	(*===================== Initializing HMI-Interface =====================*)
 	IF NOT internInstanceActivatedFirstTime THEN
		FC_InitializingSettingLines(HMIInterface := internHMIInterface);
		internInstanceActivatedFirstTime := TRUE;
	END_IF
	(*===================== Button Handling Movement =====================*)
	internHMIInterface.Movements.MovementSettingLines[1].CaptionSettingLine := CONCAT('Conveyor Control ', ActorInstanceName);
	internHMIInterface.Movements.MovementSettingLines[1].VisibilitySettingLine := TRUE;
	
	internHMIInterface.Movements.MovementSettingLines[1].SettingLineButtons[1].IsVisibleButton := TRUE;
	internHMIInterface.Movements.MovementSettingLines[1].SettingLineButtons[1].IsVisibleAxisPosition := FALSE;
	internHMIInterface.Movements.MovementSettingLines[1].SettingLineButtons[1].IsEnabled := OperatingMode.ManuelIsActive AND NOT
																							statMotorBackward AND NOT
									 														OperatingMode.EStop.IsActive AND NOT
																							statErrorRuncontrolForward;
	internHMIInterface.Movements.MovementSettingLines[1].SettingLineButtons[1].InPosition := statMotorForward;
	internHMIInterface.Movements.MovementSettingLines[1].SettingLineButtons[1].CaptionButton := 'Forward';
	internHMIInterface.Movements.MovementSettingLines[1].SettingLineButtons[1].PathImageButton := 'Images\ForwardConveyor.svg';
	
	internHMIInterface.Movements.MovementSettingLines[1].SettingLineButtons[2].IsVisibleButton := TRUE;
	internHMIInterface.Movements.MovementSettingLines[1].SettingLineButtons[2].IsVisibleAxisPosition := FALSE;
	internHMIInterface.Movements.MovementSettingLines[1].SettingLineButtons[2].IsEnabled := OperatingMode.ManuelIsActive;
	internHMIInterface.Movements.MovementSettingLines[1].SettingLineButtons[2].InPosition := NOT statMotorForward AND NOT statMotorBackward;
	internHMIInterface.Movements.MovementSettingLines[1].SettingLineButtons[2].CaptionButton := 'Stop';
	internHMIInterface.Movements.MovementSettingLines[1].SettingLineButtons[2].PathImageButton := 'Images\StopConveyor.svg';
	
	internHMIInterface.Movements.MovementSettingLines[1].SettingLineButtons[3].IsVisibleButton := TRUE;
	internHMIInterface.Movements.MovementSettingLines[1].SettingLineButtons[3].IsVisibleAxisPosition := FALSE;
	internHMIInterface.Movements.MovementSettingLines[1].SettingLineButtons[3].IsEnabled := OperatingMode.ManuelIsActive AND NOT
																							statMotorForward AND NOT
									 														OperatingMode.EStop.IsActive AND NOT
																							statErrorRuncontrolBackward;
	internHMIInterface.Movements.MovementSettingLines[1].SettingLineButtons[3].InPosition := statMotorBackward;
	internHMIInterface.Movements.MovementSettingLines[1].SettingLineButtons[3].CaptionButton := 'Backward';
	internHMIInterface.Movements.MovementSettingLines[1].SettingLineButtons[3].PathImageButton := 'Images\BackwardConveyor.svg';
	
	(*===================== Button Handling Runcontrol =====================*)
	internHMIInterface.Runcontrols.RuncontrolSettingLines[1].CaptionSettingLine := CONCAT('Runcontrol Forward ', ActorInstanceName);
	internHMIInterface.Runcontrols.RuncontrolSettingLines[1].VisibilitySettingLine := TRUE;
	
	internHMIInterface.Runcontrols.RuncontrolSettingLines[1].SettingLineButtons[1].IsVisibleButton := TRUE;
	internHMIInterface.Runcontrols.RuncontrolSettingLines[1].SettingLineButtons[1].IsVisibleAxisPosition := FALSE;
	internHMIInterface.Runcontrols.RuncontrolSettingLines[1].SettingLineButtons[1].IsEnabled := FALSE;
	internHMIInterface.Runcontrols.RuncontrolSettingLines[1].SettingLineButtons[1].InPosition := statRuncontrolForward;
	internHMIInterface.Runcontrols.RuncontrolSettingLines[1].SettingLineButtons[1].CaptionButton := 'Active';
	internHMIInterface.Runcontrols.RuncontrolSettingLines[1].SettingLineButtons[1].PathImageButton := 'Images\ActiveRuncontrol.svg';
	
	internHMIInterface.Runcontrols.RuncontrolSettingLines[1].SettingLineButtons[2].IsVisibleButton := TRUE;
	internHMIInterface.Runcontrols.RuncontrolSettingLines[1].SettingLineButtons[2].IsVisibleAxisPosition := FALSE;
	internHMIInterface.Runcontrols.RuncontrolSettingLines[1].SettingLineButtons[2].IsEnabled := statRuncontrolForward;
	internHMIInterface.Runcontrols.RuncontrolSettingLines[1].SettingLineButtons[2].InPosition := NOT statRuncontrolForward;
	internHMIInterface.Runcontrols.RuncontrolSettingLines[1].SettingLineButtons[2].CaptionButton := 'Reset';
	internHMIInterface.Runcontrols.RuncontrolSettingLines[1].SettingLineButtons[2].PathImageButton := 'Images\ResetRuncontrol.svg';
	
	internHMIInterface.Runcontrols.RuncontrolSettingLines[2].CaptionSettingLine := CONCAT('Runcontrol Backward ', ActorInstanceName);
	internHMIInterface.Runcontrols.RuncontrolSettingLines[2].VisibilitySettingLine := TRUE;
	
	internHMIInterface.Runcontrols.RuncontrolSettingLines[2].SettingLineButtons[1].IsVisibleButton := TRUE;
	internHMIInterface.Runcontrols.RuncontrolSettingLines[2].SettingLineButtons[1].IsVisibleAxisPosition := FALSE;
	internHMIInterface.Runcontrols.RuncontrolSettingLines[2].SettingLineButtons[1].IsEnabled := FALSE;
	internHMIInterface.Runcontrols.RuncontrolSettingLines[2].SettingLineButtons[1].InPosition := statRuncontrolBackward;
	internHMIInterface.Runcontrols.RuncontrolSettingLines[2].SettingLineButtons[1].CaptionButton := 'Active';
	internHMIInterface.Runcontrols.RuncontrolSettingLines[2].SettingLineButtons[1].PathImageButton := 'Images\ActiveRuncontrol.svg';
	
	internHMIInterface.Runcontrols.RuncontrolSettingLines[2].SettingLineButtons[2].IsVisibleButton := TRUE;
	internHMIInterface.Runcontrols.RuncontrolSettingLines[2].SettingLineButtons[2].IsVisibleAxisPosition := FALSE;
	internHMIInterface.Runcontrols.RuncontrolSettingLines[2].SettingLineButtons[2].IsEnabled := statRuncontrolBackward;
	internHMIInterface.Runcontrols.RuncontrolSettingLines[2].SettingLineButtons[2].InPosition := NOT statRuncontrolBackward;
	internHMIInterface.Runcontrols.RuncontrolSettingLines[2].SettingLineButtons[2].CaptionButton := 'Reset';
	internHMIInterface.Runcontrols.RuncontrolSettingLines[2].SettingLineButtons[2].PathImageButton := 'Images\ResetRuncontrol.svg';
	
	(*===================== Conveyor Forward =====================*)
	internRisingEdgePressButtonForward(CLK := internHMIInterface.Movements.MovementSettingLines[1].SettingLineButtons[1].IsPressed);
	IF(internRisingEdgePressButtonForward.Q) THEN
		statMotorForward := TRUE;
	END_IF
	(*===================== Conveyor Backward =====================*)
	internRisingEdgePressButtonBackward(CLK := internHMIInterface.Movements.MovementSettingLines[1].SettingLineButtons[3].IsPressed);
	IF(internRisingEdgePressButtonBackward.Q) THEN
		statMotorBackward := TRUE;
	END_IF
	(*===================== Conveyor Stop =====================*)
	internRisingEdgePressButtonStop(CLK := internHMIInterface.Movements.MovementSettingLines[1].SettingLineButtons[2].IsPressed);
	IF(internRisingEdgePressButtonStop.Q) THEN
		statMotorForward := FALSE;
		statMotorBackward := FALSE;
	END_IF
	(*===================== Runcontrol Forward =====================*)
	internRisingEdgePressButtonRuncontrolForwardReset(CLK := internHMIInterface.Runcontrols.RuncontrolSettingLines[1].SettingLineButtons[2].IsPressed);
	IF(internRisingEdgePressButtonRuncontrolForwardReset.Q) THEN
		internResetRuncontrolForward := TRUE;
	END_IF
	(*===================== Runcontrol Backward =====================*)
	internRisingEdgePressButtonRuncontrolBackwardReset(CLK := internHMIInterface.Runcontrols.RuncontrolSettingLines[2].SettingLineButtons[2].IsPressed);
	IF(internRisingEdgePressButtonRuncontrolBackwardReset.Q) THEN
		internResetRuncontrolBackward := TRUE;
	END_IF
	(*===================== Write Interface =====================*)
	HMIInterface := internHMIInterface;
ELSE
		internInstanceActivatedFirstTime := FALSE;
END_IF
(*===================== Motor Forward =====================*)
statMotorForward := statMotorForward AND ((OperatingMode.AutomaticIsActive
									 AND(OperatingMode.AutomaticStart.IsActive OR 
										 OperatingMode.AutomaticHome.IsActive) AND NOT
									 	 OperatingMode.AutomaticStop.IsActive) OR
										 OperatingMode.ManuelIsActive) AND NOT
										 statMotorBackward AND NOT
									 	 OperatingMode.EStop.IsActive AND NOT
										 statErrorRuncontrolForward;
(*===================== Motor Backward =====================*)
statMotorBackward := statMotorBackward AND ((OperatingMode.AutomaticIsActive
									   AND(OperatingMode.AutomaticStart.IsActive OR 
										   OperatingMode.AutomaticHome.IsActive) AND NOT
									 	   OperatingMode.AutomaticStop.IsActive) OR
											OperatingMode.ManuelIsActive) AND NOT
										   statMotorForward AND NOT
									 	   OperatingMode.EStop.IsActive AND NOT
										   statErrorRuncontrolBackward;
(*===================== Runcontrol Forward =====================*)
IF statMotorForward AND NOT statRuncontrolForward THEN
	statRuncontrolForward := TRUE;
ELSIF (statRuncontrolForward AND SensorOutfeed) OR
	(OperatingMode.ManuelIsActive AND internResetRuncontrolForward AND statErrorRuncontrolForward)
THEN
		statRuncontrolForward := FALSE;
		internResetRuncontrolForward := FALSE;
END_IF

statTimeRuncontrolForward(IN:= statRuncontrolForward,
						  PT:= MaximumTimeRuncontrol);
IF OperatingMode.Quit.IsActive THEN
	statErrorRuncontrolForward := FALSE;
END_IF
IF statTimeRuncontrolForward.Q THEN
	statErrorRuncontrolForward := TRUE;
END_IF
(*===================== Runcontrol Backward =====================*)
IF statMotorBackward AND NOT statRuncontrolBackward THEN
	statRuncontrolBackward := TRUE;
ELSIF statRuncontrolBackward AND SensorInfeed OR
	(OperatingMode.ManuelIsActive AND internResetRuncontrolBackward AND statErrorRuncontrolBackward)
THEN
		statRuncontrolBackward := FALSE;
		internResetRuncontrolBackward := FALSE;
END_IF

statTimeRuncontrolBackward(IN:= statRuncontrolBackward,
						   PT:= MaximumTimeRuncontrol);
IF OperatingMode.Quit.IsActive THEN
	statErrorRuncontrolBackward := FALSE;
END_IF
IF statTimeRuncontrolBackward.Q THEN
	statErrorRuncontrolBackward := TRUE;
END_IF
(*===================== Outputs =====================*)
MotorForward := statMotorForward;
MotorBackward := statMotorBackward;
RuncontrolForwardActive := statRuncontrolForward;
RuncontrolBackwardActive := statRuncontrolBackward;
Error := statErrorRuncontrolForward OR statErrorRuncontrolBackward;
OperatingMode.Fault.IsActive :=  statErrorRuncontrolForward OR statErrorRuncontrolBackward;

METHOD PUBLIC Motor_Off
VAR_INPUT
	Motor_Stop	:	BOOL;
END_VAR
IF Motor_Stop THEN
	statMotorForward := FALSE;
	statMotorBackward := FALSE;
END_IF
END_METHOD

METHOD MotorBackward_On
VAR_INPUT
	MotorBackward_Start	:	BOOL;
END_VAR
IF OperatingMode.AutomaticIsActive AND
(OperatingMode.AutomaticStart.IsActive OR 
 OperatingMode.AutomaticHome.IsActive) AND NOT
 statMotorForward AND NOT
 OperatingMode.AutomaticStop.IsActive AND NOT
 OperatingMode.EStop.IsActive AND NOT
 statErrorRuncontrolBackward AND NOT
 statMotorBackward AND
 MotorBackward_Start
 THEN
 	statMotorBackward := TRUE;
END_IF
END_METHOD

METHOD PUBLIC MotorForward_On
VAR_INPUT
	MotorForward_Start	:	BOOL;
END_VAR
IF  OperatingMode.AutomaticIsActive AND
(OperatingMode.AutomaticStart.IsActive OR 
 OperatingMode.AutomaticHome.IsActive) AND NOT
 statMotorBackward AND NOT
 OperatingMode.AutomaticStop.IsActive AND NOT
 OperatingMode.EStop.IsActive AND NOT
 statErrorRuncontrolForward AND NOT
 statMotorForward AND
 MotorForward_Start
 THEN
	statMotorForward := TRUE;
END_IF
END_METHOD

END_FUNCTION_BLOCK

// ---- POUs/Vorlagen/HMI/FB_HMIHeader.TcPOU
FUNCTION_BLOCK FB_HMIHeader
VAR_INPUT
	NameApplication	:	STRING;
	OperatingModeHMIInterface	:	HMIInterfaceOperatingMode;
END_VAR
VAR_OUTPUT
END_VAR
VAR_IN_OUT
	HeaderHMIInterface	:	HMIHeader;
END_VAR
VAR
	statHeaderHMIInterface	:	HMIHeader;
END_VAR

(*===================== Name Application =====================*)
statHeaderHMIInterface.NameApplication := NameApplication;
(*===================== Name Application =====================*)
statHeaderHMIInterface.ErrorIsActive := OperatingModeHMIInterface.PLCToHMI.CurrentOperatingMode.Fault.IsActive;
(*===================== Operating Mode =====================*)
IF OperatingModeHMIInterface.PLCToHMI.CurrentOperatingMode.ManuelIsActive THEN
	statHeaderHMIInterface.PathOperatingMode := 'Images/Manual_Mode.svg';
	statHeaderHMIInterface.State := 1;
ELSIF OperatingModeHMIInterface.PLCToHMI.CurrentOperatingMode.AutomaticIsActive THEN
	statHeaderHMIInterface.PathOperatingMode := 'Images/Automatic_Mode.svg';
	statHeaderHMIInterface.State := 2;
END_IF
(*===================== Operating State =====================*)
IF OperatingModeHMIInterface.PLCToHMI.CurrentOperatingMode.AutomaticStart.IsActive THEN
	statHeaderHMIInterface.PathMachineState := 'Images/Machine_Run.svg';
	statHeaderHMIInterface.State := 3;
ELSIF OperatingModeHMIInterface.PLCToHMI.CurrentOperatingMode.AutomaticStop.IsActive THEN
	statHeaderHMIInterface.PathMachineState := 'Images/Machine_Stop.svg';
	statHeaderHMIInterface.State := 2;	
ELSIF OperatingModeHMIInterface.PLCToHMI.CurrentOperatingMode.AutomaticHome.IsActive THEN
	statHeaderHMIInterface.PathMachineState := 'Images/Home-Symbol.svg';
	statHeaderHMIInterface.State := 4;			
END_IF
(*===================== Outputs =====================*)
HeaderHMIInterface := statHeaderHMIInterface;

END_FUNCTION_BLOCK

// ---- POUs/Vorlagen/Communication/ADS/FB_ADSCommunicationStatus.TcPOU
FUNCTION_BLOCK FB_ADSCommunicationStatus
VAR_INPUT
	Timeout	:	TIME := T#1S;
	TimeoutHMI	:	TIME := T#1S;
	LocalAdsPort	:	T_AmsPort := 851;
	HeartbeatHMI	:	BOOL;
END_VAR
VAR
	instReadLocalAMSNetId	:	FB_GetLocalAmsNetId;
	statExecuteReadingLocalAMSNetId	:	BOOL := TRUE;
	statBusyReadLocalAMSNetId	:	BOOL;
	statErrorReadLocalAMSNetId	:	BOOL;
	statErrorNumberReadLocalAMSNetId	:	UDINT;
	statReadLocalAMSNetId	:	T_AmsNetID;
	statReadLocalAMSNetIdSeprated	:	T_AmsNetIdArr;
	
	statGettingIpAddress	:	BOOL;
	statLocalIpAddress	:	STRING;
	
	instReadADSState	:	ADSRDSTATE;
	statExecuteReadingAdsState	:	BOOL;
	statBusyReadAdsState	:	BOOL;
	statErrorReadAdsState	:	BOOL;
	statErrorNumberAdsState	:	UDINT;
	statReadAdsState	:	UDINT;
	
	statConvertingAdsState	:	BOOL;
	statConvertedAdsState	:	STRING;
	
	instHearbeatEvaluationHMITrue	:	TON;
	instHearbeatEvaluationHMIFalse	:	TON;
	statErrorHeartbeatHMIToLongTrue	:	BOOL;
	statErrorHeartbeatHMIToLongFalse	:	BOOL;
	statHearbeatHMIIsKeepAlive	:	BOOL;
	
	instHearbeatPLCTrue	:	TON;
	instHearbeatPLCFalse	:	TON;
	statHeartbeatPLCTrue	:	BOOL;
	statHeartbeatPLCFalse	:	BOOL;
	statHearbeatPLC	:	BOOL;
END_VAR

(*===================== Reading local AMSNetId =====================*)
instReadLocalAMSNetId(bExecute := statExecuteReadingLocalAMSNetId,
					  tTimeOut := Timeout,
					  bBusy => statBusyReadLocalAMSNetId,
					  bError => statErrorReadLocalAMSNetId,
					  nErrId => statErrorNumberReadLocalAMSNetId,
					  AddrString => statReadLocalAMSNetId,
					  AddrBytes => statReadLocalAMSNetIdSeprated);
					  
IF NOT statBusyReadLocalAMSNetId AND NOT statErrorReadLocalAMSNetId AND
	statExecuteReadingLocalAMSNetId THEN
	statExecuteReadingLocalAMSNetId := FALSE;
	statGettingIpAddress := TRUE;
	statExecuteReadingAdsState := TRUE;
END_IF

(*===================== Getting IP-Address =====================*)
IF statGettingIpAddress THEN
	statLocalIpAddress := GetDeviceIpAddress(statReadLocalAMSNetIdSeprated);
	statGettingIpAddress := FALSE;
END_IF

(*===================== Reading Ads state =====================*)
instReadADSState(NETID := statReadLocalAMSNetId,
				 PORT := LocalAdsPort,
				 RDSTATE := statExecuteReadingAdsState,
			     TMOUT := Timeout,
				 BUSY => statBusyReadAdsState,
				 ERR => statErrorReadAdsState,
				 ERRID => statErrorNumberAdsState,
				 ADSSTATE => statReadAdsState);
					  
IF NOT statBusyReadAdsState AND NOT statErrorReadAdsState AND
	statExecuteReadingAdsState THEN
	statExecuteReadingAdsState := FALSE;
	statConvertingAdsState := TRUE;
END_IF

(*===================== Converting Ads state =====================*)
IF statConvertingAdsState THEN
	statConvertedAdsState := ConvertRuntimestatusInString(statReadAdsState);
	statConvertingAdsState := FALSE;
END_IF

(*===================== Evaluating Heartbeat HMI =====================*)
instHearbeatEvaluationHMITrue(IN := HeartbeatHMI,
							  PT := TimeoutHMI,
							  Q => statErrorHeartbeatHMIToLongTrue);
instHearbeatEvaluationHMIFalse(IN := NOT HeartbeatHMI,
							  PT := TimeoutHMI,
							  Q => statErrorHeartbeatHMIToLongFalse);
							  

statHearbeatHMIIsKeepAlive := NOT statErrorHeartbeatHMIToLongTrue AND NOT statErrorHeartbeatHMIToLongFalse;

(*===================== Creating Heartbeat PLC =====================*)
instHearbeatPLCTrue(IN := NOT statHeartbeatPLCFalse,
					PT := TimeoutHMI,
					Q => statHeartbeatPLCTrue);
instHearbeatPLCFalse(IN := NOT statHeartbeatPLCTrue,
					 PT := TimeoutHMI,
					 Q => statHeartbeatPLCFalse);
							  

statHearbeatPLC := statHeartbeatPLCTrue;

PROPERTY PUBLIC AdsState : String
GET
AdsState := statConvertedAdsState;
END_GET
END_PROPERTY

METHOD PRIVATE ConvertRuntimestatusInString : String
VAR_INPUT
	CurrentDeviceStatus 	: 	UDINT;
END_VAR
VAR
	tempConvertedDeviceStatus	:	STRING;
END_VAR
CASE CurrentDeviceStatus OF
	0:
		tempConvertedDeviceStatus := 'Invalid';
	1:
		tempConvertedDeviceStatus := 'Idle';
	2:
		tempConvertedDeviceStatus := 'Reset';
	3:
		tempConvertedDeviceStatus := 'Init';
	4:
		tempConvertedDeviceStatus := 'Start';
	5:
		tempConvertedDeviceStatus := 'Run';
	6:
		tempConvertedDeviceStatus := 'Stop';
	7:
		tempConvertedDeviceStatus := 'Save cfg';
	8:
		tempConvertedDeviceStatus := 'Load cfg';
	9:
		tempConvertedDeviceStatus := 'Power failure';
	10:
		tempConvertedDeviceStatus := 'Power good';
	11:
		tempConvertedDeviceStatus := 'Error';
	12:
		tempConvertedDeviceStatus := 'Shutdown';
	13:
		tempConvertedDeviceStatus := 'Suspend';
	14:
		tempConvertedDeviceStatus := 'Resume';
	15:
		tempConvertedDeviceStatus := 'Config';
	16:
		tempConvertedDeviceStatus := 'Reconfig';
	17:
		tempConvertedDeviceStatus := 'Stopping';
	18:
		tempConvertedDeviceStatus := 'Incompatible';
	19:
		tempConvertedDeviceStatus := 'Execption';
	ELSE
		tempConvertedDeviceStatus := 'Not defined in system';			
END_CASE

ConvertRuntimestatusInString := tempConvertedDeviceStatus;
END_METHOD

METHOD PRIVATE GetDeviceIpAddress : String
VAR_INPUT
	CurrentAMSNetId	:	T_AmsNetIdArr;
END_VAR
VAR
	tempRunCounter	:	INT;
	tempIpAddressConverted	:	STRING;
END_VAR
FOR tempRunCounter := 0 TO 3 DO
	tempIpAddressConverted := CONCAT(tempIpAddressConverted, BYTE_TO_STRING(CurrentAMSNetId[tempRunCounter]));
	IF tempRunCounter < 3 THEN
		tempIpAddressConverted := CONCAT(tempIpAddressConverted, '.');
	END_IF
END_FOR

GetDeviceIpAddress := tempIpAddressConverted;
END_METHOD

PROPERTY PUBLIC HMICommunicationIsActive : BOOL
GET
HMICommunicationIsActive := statHearbeatHMIIsKeepAlive;
END_GET
END_PROPERTY

PROPERTY PUBLIC LocalAMSNetId : String
GET
LocalAMSNetId := statReadLocalAMSNetId;
END_GET
END_PROPERTY

PROPERTY PUBLIC LocalIpAddress : String
GET
LocalIpAddress := statLocalIpAddress;
END_GET
END_PROPERTY

PROPERTY PUBLIC PLCHeartbeatHMICommunication : BOOL
GET
PLCHeartbeatHMICommunication := statHearbeatPLC;
END_GET
END_PROPERTY

END_FUNCTION_BLOCK

// ---- POUs/Vorlagen/PickPlace/FB_PickPlace_DigitalAnalog.TcPOU
FUNCTION_BLOCK FB_PickPlace_DigitalAnalog
VAR_INPUT
	PickPlaceCurrentPositionXAxis	:	WORD;	//Raw value X axis
	PickPlaceCurrentPositionYAxis	:	WORD;	//Raw value Y axis
	PickPlaceCurrentPositionZAxis	:	WORD;	//Raw value Z axis
	PickPlaceX_YAxisStillMoving	:	BOOL;	//X and Y axis are moving
	PickPlaceZAxisStillMoving	:	BOOL;	//Z axis are moving
	PickPlaceBoxDetected	:	BOOL;	//Box detected on Gripper
	PickPlaceCAxisLimitReached	:	BOOL;	//C axis in Position
	ActorInstanceIndex	:	INT;	//Index in DropDown HMI
	ActorInstanceName	:	STRING;		//Name of the instance
END_VAR
VAR_OUTPUT
	SetPointToXAxis : WORD;	//Setpoint X axis
	SetPointToYAxis : WORD;	//Setpoint Y axis
	SetPointToZAxis : WORD;	//Setpoint Z axis
	GrabPart	:	BOOL;	//Grab a part
	RotateGripper	:	BOOL;	//Rotate gripper
END_VAR
VAR_IN_OUT
	OperatingMode	:	OperatingMode;	//Schnittstelle für Betriebsarten
	HMIInterface	:	MachineSectionHMIInterface;	//HMI-Interface
END_VAR
VAR
	statInit	:	BOOL; //Memory for first cycle
	statMovePickPlace	:	BOOL;
	statPickPlaceNewOrder	:	BOOL;
	statPickPlaceInPositionXAxis	:	BOOL := TRUE;
	statPickPlaceInPositionYAxis	:	BOOL := TRUE;
	statPickPlaceInPositionZAxis	:	BOOL := TRUE;
	statPickPlaceInPositionCAxis90	:	BOOL;
	statCurrentPositionXAxis	: REAL;
	statCurrentPositionYAxis	: REAL;
	statCurrentPositionZAxis	: REAL;
	statSelectedSetPointXAxis	: REAL;
	statSelectedSetPointYAxis	: REAL;
	statSelectedSetPointZAxis	: REAL;
	statSetPointXAxis	:	REAL;
	statSetPointYAxis	:	REAL;
	statSetPointZAxis	:	REAL;
	statSetPointToXaxis	:	WORD;
	statSetPointToYaxis	:	WORD;
	statSetPointToZaxis	:	WORD;
	statCAxisToPos90	:	BOOL;
	statGrabPart	:	BOOL;
	statREX_YAxisMoving	:	R_TRIG;
	statREZAxisMoving	:	R_TRIG;
	statRECAxisMoving	:	R_TRIG;
	statFEX_YAxisMoving	:	F_TRIG;
	statFEZAxisMoving	:	F_TRIG;
	statFECAxisMoving	:	F_TRIG;
	
	internHMIInterface	:	MachineSectionHMIInterface;
	internInstanceActivatedFirstTime	:	BOOL;
	internRisingEdgePageSwitchUp	:	R_TRIG;
	internRisingEdgePageSwitchDown	:	R_TRIG;
	internRisingEdgePressButtonPlusXAxis	:	R_TRIG;
	internRisingEdgePressButtonMinusXAxis	:	R_TRIG;
	internRisingEdgePressButtonStopXAxis	:	R_TRIG;
	internRisingEdgePressButtonPlusYAxis	:	R_TRIG;
	internRisingEdgePressButtonMinusYAxis	:	R_TRIG;
	internRisingEdgePressButtonStopYAxis	:	R_TRIG;
	internRisingEdgePressButtonUpZAxis	:	R_TRIG;
	internRisingEdgePressButtonDownZAxis	:	R_TRIG;
	internRisingEdgePressButtonStopZAxis	:	R_TRIG;
	internRisingEdgePressButtonCAxisToPos90	:	R_TRIG;
	internRisingEdgePressButtonCAxisToPos0	:	R_TRIG;
	internRisingEdgePressButtonGrabPart	:	R_TRIG;
	internRisingEdgePressButtonReleasePart	:	R_TRIG;
	internStopXAxis	:	BOOL;
	internStopYAxis	:	BOOL;
	internStopZAxis	:	BOOL;
END_VAR

(*===================== CurrentPosition Axes =====================*)
FC_AnalogInputValueHandling(RowValue:= PickPlaceCurrentPositionXAxis, 
							UpperLimit:= 2.125, 
							LowerLimit:= 0.0, 
							ConvertedValue=> statCurrentPositionXAxis);
FC_AnalogInputValueHandling(RowValue:= PickPlaceCurrentPositionYAxis, 
							UpperLimit:= 1.25, 
							LowerLimit:= 0.0, 
							ConvertedValue=> statCurrentPositionYAxis);
FC_AnalogInputValueHandling(RowValue:= PickPlaceCurrentPositionZAxis, 
							UpperLimit:= 0.5, 
							LowerLimit:= 0.0, 
							ConvertedValue=> statCurrentPositionZAxis);
(*===================== HMI INTERFACE =====================*)
internHMIInterface := HMIInterface;

IF internHMIInterface.ActiveMachineSection = MachineSection.PickPlace AND
	internHMIInterface.SelectedActor = ActorInstanceIndex THEN
	(*===================== Initializing HMI-Interface =====================*)
	IF NOT internInstanceActivatedFirstTime THEN
		FC_InitializingSettingLines(HMIInterface := internHMIInterface);
		internInstanceActivatedFirstTime := TRUE;
	END_IF
	(*===================== Page switch =====================*)
	internRisingEdgePageSwitchUp(CLK := internHMIInterface.PageSwitch.NextPageIsPressed);
	internRisingEdgePageSwitchDown(CLK := internHMIInterface.PageSwitch.PreviousPageIsPressed);
	IF internRisingEdgePageSwitchUp.Q THEN
		internHMIInterface.PageSwitch.SelectedPage := internHMIInterface.PageSwitch.SelectedPage + 1; 
	END_IF
	IF internRisingEdgePageSwitchDown.Q THEN
		internHMIInterface.PageSwitch.SelectedPage := internHMIInterface.PageSwitch.SelectedPage - 1; 
	END_IF
	IF internHMIInterface.PageSwitch.SelectedPage = 0 THEN
		internHMIInterface.PageSwitch.SelectedPage := 1;
	END_IF
	internHMIInterface.PageSwitch.MinPage := 1;
	internHMIInterface.PageSwitch.MaxPage := 2;
	internHMIInterface.PageSwitch.NextPageIsEnabled := internHMIInterface.PageSwitch.SelectedPage < internHMIInterface.PageSwitch.MaxPage;
	internHMIInterface.PageSwitch.PreviousPageIsEnabled := internHMIInterface.PageSwitch.SelectedPage > internHMIInterface.PageSwitch.MinPage;
	(*===================== Button Handling Movement =====================*)
	IF internHMIInterface.PageSwitch.SelectedPage = 1 THEN
		internHMIInterface.Movements.MovementSettingLines[1].CaptionSettingLine := CONCAT('StackerCrane X-Axis Control ', ActorInstanceName);
		internHMIInterface.Movements.MovementSettingLines[1].VisibilitySettingLine := TRUE;
		
		internHMIInterface.Movements.MovementSettingLines[1].SettingLineButtons[1].IsVisibleButton := TRUE;
		internHMIInterface.Movements.MovementSettingLines[1].SettingLineButtons[1].IsVisibleAxisPosition := FALSE;
		internHMIInterface.Movements.MovementSettingLines[1].SettingLineButtons[1].IsEnabled := OperatingMode.ManuelIsActive AND NOT
										 														OperatingMode.EStop.IsActive AND NOT
																								OperatingMode.Fault.IsActive AND NOT
																								statMovePickPlace AND
																								statSetPointXAxis < 2.215;
		internHMIInterface.Movements.MovementSettingLines[1].SettingLineButtons[1].InPosition := statPickPlaceInPositionXAxis;
		internHMIInterface.Movements.MovementSettingLines[1].SettingLineButtons[1].CaptionButton := 'Plus';
		internHMIInterface.Movements.MovementSettingLines[1].SettingLineButtons[1].PathImageButton := 'Images\ForwardConveyor.svg';
		
		internHMIInterface.Movements.MovementSettingLines[1].SettingLineButtons[2].IsVisibleButton := TRUE;
		internHMIInterface.Movements.MovementSettingLines[1].SettingLineButtons[2].IsVisibleAxisPosition := TRUE;
		internHMIInterface.Movements.MovementSettingLines[1].SettingLineButtons[2].IsEnabled := OperatingMode.ManuelIsActive;
		internHMIInterface.Movements.MovementSettingLines[1].SettingLineButtons[2].InPosition := NOT statMovePickPlace;
		internHMIInterface.Movements.MovementSettingLines[1].SettingLineButtons[2].AxisPosition := statCurrentPositionXAxis;
		internHMIInterface.Movements.MovementSettingLines[1].SettingLineButtons[2].CaptionButton := 'Stop';
		internHMIInterface.Movements.MovementSettingLines[1].SettingLineButtons[2].PathImageButton := 'Images\StopConveyor.svg';
		
		internHMIInterface.Movements.MovementSettingLines[1].SettingLineButtons[3].IsVisibleButton := TRUE;
		internHMIInterface.Movements.MovementSettingLines[1].SettingLineButtons[3].IsVisibleAxisPosition := FALSE;
		internHMIInterface.Movements.MovementSettingLines[1].SettingLineButtons[3].IsEnabled := OperatingMode.ManuelIsActive AND NOT
										 														OperatingMode.EStop.IsActive AND NOT
																								OperatingMode.Fault.IsActive AND NOT
																								statMovePickPlace AND
																								statSetPointXAxis > 0.1;
		internHMIInterface.Movements.MovementSettingLines[1].SettingLineButtons[3].InPosition := statPickPlaceInPositionXAxis;
		internHMIInterface.Movements.MovementSettingLines[1].SettingLineButtons[3].CaptionButton := 'Minus';
		internHMIInterface.Movements.MovementSettingLines[1].SettingLineButtons[3].PathImageButton := 'Images\BackwardConveyor.svg';
		
		internHMIInterface.Movements.MovementSettingLines[2].CaptionSettingLine := CONCAT('StackerCrane Y-Axis Control ', ActorInstanceName);
		internHMIInterface.Movements.MovementSettingLines[2].VisibilitySettingLine := TRUE;
		
		internHMIInterface.Movements.MovementSettingLines[2].SettingLineButtons[1].IsVisibleButton := TRUE;
		internHMIInterface.Movements.MovementSettingLines[2].SettingLineButtons[1].IsVisibleAxisPosition := FALSE;
		internHMIInterface.Movements.MovementSettingLines[2].SettingLineButtons[1].IsEnabled := OperatingMode.ManuelIsActive AND NOT
										 														OperatingMode.EStop.IsActive AND NOT
																								OperatingMode.Fault.IsActive AND NOT
																								statMovePickPlace AND
																								statSetPointYAxis < 1.25;
		internHMIInterface.Movements.MovementSettingLines[2].SettingLineButtons[1].InPosition := statPickPlaceInPositionYAxis;
		internHMIInterface.Movements.MovementSettingLines[2].SettingLineButtons[1].CaptionButton := 'Plus';
		internHMIInterface.Movements.MovementSettingLines[2].SettingLineButtons[1].PathImageButton := 'Images\UpElevator.svg';
		
		internHMIInterface.Movements.MovementSettingLines[2].SettingLineButtons[2].IsVisibleButton := TRUE;
		internHMIInterface.Movements.MovementSettingLines[2].SettingLineButtons[2].IsVisibleAxisPosition := TRUE;
		internHMIInterface.Movements.MovementSettingLines[2].SettingLineButtons[2].IsEnabled := OperatingMode.ManuelIsActive;
		internHMIInterface.Movements.MovementSettingLines[2].SettingLineButtons[2].InPosition := NOT statMovePickPlace;
		internHMIInterface.Movements.MovementSettingLines[2].SettingLineButtons[2].AxisPosition := statCurrentPositionYAxis;
		internHMIInterface.Movements.MovementSettingLines[2].SettingLineButtons[2].CaptionButton := 'Stop';
		internHMIInterface.Movements.MovementSettingLines[2].SettingLineButtons[2].PathImageButton := 'Images\StopConveyor.svg';
		
		internHMIInterface.Movements.MovementSettingLines[2].SettingLineButtons[3].IsVisibleButton := TRUE;
		internHMIInterface.Movements.MovementSettingLines[2].SettingLineButtons[3].IsVisibleAxisPosition := FALSE;
		internHMIInterface.Movements.MovementSettingLines[2].SettingLineButtons[3].IsEnabled := OperatingMode.ManuelIsActive AND NOT
										 														OperatingMode.EStop.IsActive AND NOT
																								OperatingMode.Fault.IsActive AND NOT
																								statMovePickPlace AND
																								statSetPointYAxis > 0.1;
		internHMIInterface.Movements.MovementSettingLines[2].SettingLineButtons[3].InPosition := statPickPlaceInPositionYAxis;
		internHMIInterface.Movements.MovementSettingLines[2].SettingLineButtons[3].CaptionButton := 'Minus';
		internHMIInterface.Movements.MovementSettingLines[2].SettingLineButtons[3].PathImageButton := 'Images\DownElevator.svg';
	
	ELSIF internHMIInterface.PageSwitch.SelectedPage = 2 THEN
		internHMIInterface.Movements.MovementSettingLines[1].CaptionSettingLine := CONCAT('StackerCrane Z-Axis Control ', ActorInstanceName);
		internHMIInterface.Movements.MovementSettingLines[1].VisibilitySettingLine := TRUE;
		
		internHMIInterface.Movements.MovementSettingLines[1].SettingLineButtons[1].IsVisibleButton := TRUE;
		internHMIInterface.Movements.MovementSettingLines[1].SettingLineButtons[1].IsVisibleAxisPosition := FALSE;
		internHMIInterface.Movements.MovementSettingLines[1].SettingLineButtons[1].IsEnabled := OperatingMode.ManuelIsActive AND NOT
										 														OperatingMode.EStop.IsActive AND NOT
																								OperatingMode.Fault.IsActive AND NOT
																								statMovePickPlace AND
																								statSetPointZAxis > 0.1;
		internHMIInterface.Movements.MovementSettingLines[1].SettingLineButtons[1].InPosition := statPickPlaceInPositionZAxis;
		internHMIInterface.Movements.MovementSettingLines[1].SettingLineButtons[1].CaptionButton := 'Up';
		internHMIInterface.Movements.MovementSettingLines[1].SettingLineButtons[1].PathImageButton := 'Images\UpElevator.svg';
		
		internHMIInterface.Movements.MovementSettingLines[1].SettingLineButtons[2].IsVisibleButton := TRUE;
		internHMIInterface.Movements.MovementSettingLines[1].SettingLineButtons[2].IsVisibleAxisPosition := TRUE;
		internHMIInterface.Movements.MovementSettingLines[1].SettingLineButtons[2].IsEnabled := OperatingMode.ManuelIsActive;
		internHMIInterface.Movements.MovementSettingLines[1].SettingLineButtons[2].InPosition := NOT statMovePickPlace;
		internHMIInterface.Movements.MovementSettingLines[1].SettingLineButtons[2].AxisPosition := statCurrentPositionZAxis;
		internHMIInterface.Movements.MovementSettingLines[1].SettingLineButtons[2].CaptionButton := 'Stop';
		internHMIInterface.Movements.MovementSettingLines[1].SettingLineButtons[2].PathImageButton := 'Images\StopConveyor.svg';
		
		internHMIInterface.Movements.MovementSettingLines[1].SettingLineButtons[3].IsVisibleButton := TRUE;
		internHMIInterface.Movements.MovementSettingLines[1].SettingLineButtons[3].IsVisibleAxisPosition := FALSE;
		internHMIInterface.Movements.MovementSettingLines[1].SettingLineButtons[3].IsEnabled := OperatingMode.ManuelIsActive AND NOT
										 														OperatingMode.EStop.IsActive AND NOT
																								OperatingMode.Fault.IsActive AND NOT
																								statMovePickPlace AND
																								statSetPointZAxis < 0.5;
		internHMIInterface.Movements.MovementSettingLines[1].SettingLineButtons[3].InPosition := statPickPlaceInPositionZAxis;
		internHMIInterface.Movements.MovementSettingLines[1].SettingLineButtons[3].CaptionButton := 'Down';
		internHMIInterface.Movements.MovementSettingLines[1].SettingLineButtons[3].PathImageButton := 'Images\DownElevator.svg';
		
		internHMIInterface.Movements.MovementSettingLines[2].CaptionSettingLine := CONCAT('StackerCrane C-Axis Control ', ActorInstanceName);
		internHMIInterface.Movements.MovementSettingLines[2].VisibilitySettingLine := TRUE;
		
		internHMIInterface.Movements.MovementSettingLines[2].SettingLineButtons[1].IsVisibleButton := TRUE;
		internHMIInterface.Movements.MovementSettingLines[2].SettingLineButtons[1].IsVisibleAxisPosition := FALSE;
		internHMIInterface.Movements.MovementSettingLines[2].SettingLineButtons[1].IsEnabled := OperatingMode.ManuelIsActive AND NOT
										 														OperatingMode.EStop.IsActive AND NOT
																								OperatingMode.Fault.IsActive AND NOT
																								statMovePickPlace;
		internHMIInterface.Movements.MovementSettingLines[2].SettingLineButtons[1].InPosition := statPickPlaceInPositionCAxis90;
		internHMIInterface.Movements.MovementSettingLines[2].SettingLineButtons[1].CaptionButton := '90°';
		internHMIInterface.Movements.MovementSettingLines[2].SettingLineButtons[1].PathImageButton := '';
		
		internHMIInterface.Movements.MovementSettingLines[2].SettingLineButtons[2].IsVisibleButton := FALSE;
		internHMIInterface.Movements.MovementSettingLines[2].SettingLineButtons[2].IsVisibleAxisPosition := FALSE;
		internHMIInterface.Movements.MovementSettingLines[2].SettingLineButtons[2].IsEnabled := FALSE;
		internHMIInterface.Movements.MovementSettingLines[2].SettingLineButtons[2].InPosition := FALSE;
		internHMIInterface.Movements.MovementSettingLines[2].SettingLineButtons[2].AxisPosition := 0;
		internHMIInterface.Movements.MovementSettingLines[2].SettingLineButtons[2].CaptionButton := '';
		internHMIInterface.Movements.MovementSettingLines[2].SettingLineButtons[2].PathImageButton := '';
		
		internHMIInterface.Movements.MovementSettingLines[2].SettingLineButtons[3].IsVisibleButton := TRUE;
		internHMIInterface.Movements.MovementSettingLines[2].SettingLineButtons[3].IsVisibleAxisPosition := FALSE;
		internHMIInterface.Movements.MovementSettingLines[2].SettingLineButtons[3].IsEnabled := OperatingMode.ManuelIsActive AND NOT
										 														OperatingMode.EStop.IsActive AND NOT
																								OperatingMode.Fault.IsActive AND NOT
																								statMovePickPlace;
		internHMIInterface.Movements.MovementSettingLines[2].SettingLineButtons[3].InPosition := NOT statPickPlaceInPositionCAxis90;
		internHMIInterface.Movements.MovementSettingLines[2].SettingLineButtons[3].CaptionButton := '0°';
		internHMIInterface.Movements.MovementSettingLines[2].SettingLineButtons[3].PathImageButton := '';	
		END_IF
		
		internHMIInterface.Forks.ForkMovementSettingLines[1].CaptionSettingLine := CONCAT('Fork Control ', ActorInstanceName);
		internHMIInterface.Forks.ForkMovementSettingLines[1].VisibilitySettingLine := TRUE;
		
		internHMIInterface.Forks.ForkMovementSettingLines[1].SettingLineButtons[1].IsVisibleButton := TRUE;
		internHMIInterface.Forks.ForkMovementSettingLines[1].SettingLineButtons[1].IsVisibleAxisPosition := FALSE;
		internHMIInterface.Forks.ForkMovementSettingLines[1].SettingLineButtons[1].IsEnabled := OperatingMode.ManuelIsActive AND NOT
										 														OperatingMode.EStop.IsActive AND NOT
																								OperatingMode.Fault.IsActive AND NOT
																								statMovePickPlace AND
																								statPickPlaceInPositionXAxis AND
																								statPickPlaceInPositionYAxis AND
																								statPickPlaceInPositionZAxis;
		internHMIInterface.Forks.ForkMovementSettingLines[1].SettingLineButtons[1].InPosition := FALSE;
		internHMIInterface.Forks.ForkMovementSettingLines[1].SettingLineButtons[1].CaptionButton := 'Grap';
		internHMIInterface.Forks.ForkMovementSettingLines[1].SettingLineButtons[1].PathImageButton := '';
		
		internHMIInterface.Forks.ForkMovementSettingLines[1].SettingLineButtons[2].IsVisibleButton := FALSE;
		internHMIInterface.Forks.ForkMovementSettingLines[1].SettingLineButtons[2].IsVisibleAxisPosition := FALSE;
		internHMIInterface.Forks.ForkMovementSettingLines[1].SettingLineButtons[2].IsEnabled := FALSE;
		internHMIInterface.Forks.ForkMovementSettingLines[1].SettingLineButtons[2].InPosition := FALSE;
		internHMIInterface.Forks.ForkMovementSettingLines[1].SettingLineButtons[2].CaptionButton := '';
		internHMIInterface.Forks.ForkMovementSettingLines[1].SettingLineButtons[2].PathImageButton := '';
		
		internHMIInterface.Forks.ForkMovementSettingLines[1].SettingLineButtons[3].IsVisibleButton := TRUE;
		internHMIInterface.Forks.ForkMovementSettingLines[1].SettingLineButtons[3].IsVisibleAxisPosition := FALSE;
		internHMIInterface.Forks.ForkMovementSettingLines[1].SettingLineButtons[3].IsEnabled := OperatingMode.ManuelIsActive AND NOT
										 														OperatingMode.EStop.IsActive AND NOT
																								OperatingMode.Fault.IsActive AND NOT
																								statMovePickPlace AND
																								statPickPlaceInPositionXAxis AND
																								statPickPlaceInPositionYAxis AND
																								statPickPlaceInPositionZAxis;
		internHMIInterface.Forks.ForkMovementSettingLines[1].SettingLineButtons[3].InPosition := FALSE;
		internHMIInterface.Forks.ForkMovementSettingLines[1].SettingLineButtons[3].CaptionButton := 'Release';
		internHMIInterface.Forks.ForkMovementSettingLines[1].SettingLineButtons[3].PathImageButton := '';
	
	(*===================== X-Axis Plus =====================*)
	internRisingEdgePressButtonPlusXAxis(CLK := internHMIInterface.Movements.MovementSettingLines[1].SettingLineButtons[1].IsPressed AND 
												internHMIInterface.PageSwitch.SelectedPage = 1 AND 
												internHMIInterface.PageSwitch.SelectedTab = 'tbMovement');
	IF internRisingEdgePressButtonPlusXAxis.Q THEN
		statSetPointXAxis := statSetPointXAxis + 0.2;
		statMovePickPlace := TRUE;
		statPickPlaceNewOrder := TRUE;
	END_IF
	(*===================== X-Axis Minus =====================*)
	internRisingEdgePressButtonMinusXAxis(CLK := internHMIInterface.Movements.MovementSettingLines[1].SettingLineButtons[3].IsPressed AND 
												internHMIInterface.PageSwitch.SelectedPage = 1 AND 
												internHMIInterface.PageSwitch.SelectedTab = 'tbMovement');
	IF internRisingEdgePressButtonMinusXAxis.Q THEN
		statSetPointXAxis := statSetPointXAxis - 0.2;
		statMovePickPlace := TRUE;
		statPickPlaceNewOrder := TRUE;
	END_IF
	(*===================== X-Axis Stop =====================*)
	internRisingEdgePressButtonStopXAxis(CLK := internHMIInterface.Movements.MovementSettingLines[1].SettingLineButtons[2].IsPressed AND 
												internHMIInterface.PageSwitch.SelectedPage = 1 AND 
												internHMIInterface.PageSwitch.SelectedTab = 'tbMovement');
	IF internRisingEdgePressButtonStopXAxis.Q THEN
		internStopXAxis := TRUE;
	END_IF
	(*===================== Y-Axis Plus =====================*)
	internRisingEdgePressButtonPlusYAxis(CLK := internHMIInterface.Movements.MovementSettingLines[2].SettingLineButtons[1].IsPressed AND 
												internHMIInterface.PageSwitch.SelectedPage = 1 AND 
												internHMIInterface.PageSwitch.SelectedTab = 'tbMovement');
	IF internRisingEdgePressButtonPlusYAxis.Q THEN
		statSetPointYAxis := statSetPointYAxis + 0.2;
		statMovePickPlace := TRUE;
		statPickPlaceNewOrder := TRUE;
	END_IF
	(*===================== Y-Axis Minus =====================*)
	internRisingEdgePressButtonMinusYAxis(CLK := internHMIInterface.Movements.MovementSettingLines[2].SettingLineButtons[3].IsPressed AND 
												internHMIInterface.PageSwitch.SelectedPage = 1 AND 
												internHMIInterface.PageSwitch.SelectedTab = 'tbMovement');
	IF internRisingEdgePressButtonMinusYAxis.Q THEN
		statSetPointYAxis := statSetPointYAxis - 0.2;
		statMovePickPlace := TRUE;
		statPickPlaceNewOrder := TRUE;
	END_IF
	(*===================== Y-Axis Stop =====================*)
	internRisingEdgePressButtonStopYAxis(CLK := internHMIInterface.Movements.MovementSettingLines[2].SettingLineButtons[2].IsPressed AND 
												internHMIInterface.PageSwitch.SelectedPage = 1 AND 
												internHMIInterface.PageSwitch.SelectedTab = 'tbMovement');
	IF internRisingEdgePressButtonStopYAxis.Q THEN
		internStopYAxis := TRUE;
	END_IF
	(*===================== Z-Axis Up =====================*)
	internRisingEdgePressButtonUpZAxis(CLK := internHMIInterface.Movements.MovementSettingLines[1].SettingLineButtons[1].IsPressed AND 
												internHMIInterface.PageSwitch.SelectedPage = 2 AND 
												internHMIInterface.PageSwitch.SelectedTab = 'tbMovement');
	IF internRisingEdgePressButtonUpZAxis.Q THEN
		statSetPointZAxis := statSetPointZAxis - 0.2;
		statMovePickPlace := TRUE;
		statPickPlaceNewOrder := TRUE;
	END_IF
	(*===================== Z-Axis Down =====================*)
	internRisingEdgePressButtonDownZAxis(CLK := internHMIInterface.Movements.MovementSettingLines[1].SettingLineButtons[3].IsPressed AND 
												internHMIInterface.PageSwitch.SelectedPage = 2 AND 
												internHMIInterface.PageSwitch.SelectedTab = 'tbMovement');
	IF internRisingEdgePressButtonDownZAxis.Q THEN
		statSetPointZAxis := statSetPointZAxis + 0.2;
		statMovePickPlace := TRUE;
		statPickPlaceNewOrder := TRUE;
	END_IF
	(*===================== Z-Axis Stop =====================*)
	internRisingEdgePressButtonStopZAxis(CLK := internHMIInterface.Movements.MovementSettingLines[1].SettingLineButtons[2].IsPressed AND 
												internHMIInterface.PageSwitch.SelectedPage = 2 AND 
												internHMIInterface.PageSwitch.SelectedTab = 'tbMovement');
	IF internRisingEdgePressButtonStopZAxis.Q THEN
		internStopZAxis := TRUE;
	END_IF
	(*===================== C-Axis To 90 =====================*)
	internRisingEdgePressButtonCAxisToPos90(CLK := internHMIInterface.Movements.MovementSettingLines[2].SettingLineButtons[1].IsPressed AND 
												internHMIInterface.PageSwitch.SelectedPage = 2 AND 
												internHMIInterface.PageSwitch.SelectedTab = 'tbMovement');
	IF internRisingEdgePressButtonCAxisToPos90.Q THEN
		statCAxisToPos90 := TRUE;
	END_IF
	(*===================== C-Axis To 0 =====================*)
	internRisingEdgePressButtonCAxisToPos0(CLK := internHMIInterface.Movements.MovementSettingLines[2].SettingLineButtons[3].IsPressed AND 
												internHMIInterface.PageSwitch.SelectedPage = 2 AND 
												internHMIInterface.PageSwitch.SelectedTab = 'tbMovement');
	IF internRisingEdgePressButtonCAxisToPos0.Q THEN
		statCAxisToPos90 := FALSE;
	END_IF
	(*===================== Grab Part =====================*)
	internRisingEdgePressButtonGrabPart(CLK := internHMIInterface.Forks.ForkMovementSettingLines[1].SettingLineButtons[1].IsPressed);
	IF internRisingEdgePressButtonGrabPart.Q THEN
		statGrabPart := TRUE;
	END_IF
	(*===================== Release Part =====================*)
	internRisingEdgePressButtonReleasePart(CLK := internHMIInterface.Forks.ForkMovementSettingLines[1].SettingLineButtons[3].IsPressed);
	IF internRisingEdgePressButtonReleasePart.Q THEN
		statGrabPart := FALSE;
	END_IF
	(*===================== Write Interface =====================*)
	HMIInterface := internHMIInterface;
ELSE
		internInstanceActivatedFirstTime := FALSE;
END_IF
(*===================== Stacker crane in Position =====================*)
statREX_YAxisMoving(CLK := PickPlaceX_YAxisStillMoving);
statFEX_YAxisMoving(CLK := PickPlaceX_YAxisStillMoving);
statREZAxisMoving(CLK := PickPlaceZAxisStillMoving);
statFEZAxisMoving(CLK := PickPlaceZAxisStillMoving);
statRECAxisMoving(CLK := PickPlaceCAxisLimitReached);
statFECAxisMoving(CLK := PickPlaceCAxisLimitReached);

IF statPickPlaceInPositionXAxis AND statPickPlaceInPositionYAxis AND
 statPickPlaceInPositionZAxis AND NOT statPickPlaceNewOrder
THEN
	statMovePickPlace := FALSE;
END_IF
IF statREX_YAxisMoving.Q THEN
	statPickPlaceInPositionXAxis := FALSE;
	statPickPlaceInPositionYAxis := FALSE;
	statPickPlaceNewOrder := FALSE;
END_IF
IF statFEX_YAxisMoving.Q THEN
	statPickPlaceInPositionXAxis := TRUE;
	statPickPlaceInPositionYAxis := TRUE;
END_IF
IF statREZAxisMoving.Q THEN
	statPickPlaceInPositionZAxis := FALSE;
	statPickPlaceNewOrder := FALSE;
END_IF
IF statFEZAxisMoving.Q THEN
	statPickPlaceInPositionZAxis := TRUE;
END_IF
IF statRECAxisMoving.Q THEN
	statPickPlaceInPositionCAxis90 := TRUE;
END_IF
IF statFECAxisMoving.Q THEN
	statPickPlaceInPositionCAxis90 := FALSE;
END_IF
IF NOT statInit THEN
	statPickPlaceInPositionCAxis90 := FALSE;
	statInit := TRUE;
END_IF
(*===================== Positioning Stacker crane =====================*)
IF ((OperatingMode.AutomaticIsActive AND OperatingMode.AutomaticStart.IsActive) OR
	(OperatingMode.ManuelIsActive)) 
   AND statMovePickPlace 
THEN
	statSelectedSetPointXAxis := statSetPointXAxis;
	statSelectedSetPointYAxis := statSetPointYAxis;
	statSelectedSetPointZAxis := statSetPointZAxis;
END_IF
IF OperatingMode.EStop.IsActive OR OperatingMode.Fault.IsActive OR 
((OperatingMode.AutomaticIsActive AND OperatingMode.AutomaticStop.IsActive) OR
(OperatingMode.ManuelIsActive AND (internStopXAxis OR internStopZAxis)))
THEN
	statSelectedSetPointXAxis := statCurrentPositionXAxis;
	statSelectedSetPointYAxis := statCurrentPositionYAxis;
	statSelectedSetPointZAxis := statCurrentPositionZAxis;
	statMovePickPlace := FALSE;
	internStopXAxis := FALSE;
END_IF
(*===================== SetPoint X-Axis =====================*)
FC_AnalogOutputValueHandling(Setpoint:= statSelectedSetPointXAxis, 
						     UpperLimit:= 2.125, 
							 LowerLimit:= 0.0, 
							 ConvertedValue=> statSetPointToXaxis);
(*===================== SetPoint Y-Axis =====================*)
FC_AnalogOutputValueHandling(Setpoint:= statSelectedSetPointYAxis, 
						     UpperLimit:= 1.25, 
							 LowerLimit:= 0.0, 
							 ConvertedValue=> statSetPointToYaxis);
(*===================== SetPoint Z-Axis =====================*)
FC_AnalogOutputValueHandling(Setpoint:= statSelectedSetPointZAxis, 
						     UpperLimit:= 0.5, 
							 LowerLimit:= 0.0, 
							 ConvertedValue=> statSetPointToZaxis);
(*===================== Outputs writting =====================*)
SetPointToXAxis := statSetPointToXaxis;
SetPointToYAxis := statSetPointToYaxis;
SetPointToZAxis := statSetPointToZaxis;
GrabPart := statGrabPart;
RotateGripper := statCAxisToPos90;

METHOD PUBLIC GrabPart_ON : BOOL
VAR_INPUT
	StartGrabPart	:	BOOL;
END_VAR
IF OperatingMode.AutomaticIsActive AND OperatingMode.AutomaticStart.IsActive AND
	InPositionX_Y_Axis AND InPositionZAxis AND StartGrabPart AND NOT statMovePickPlace 
THEN
	statGrabPart := TRUE;
	GrabPart_ON := TRUE;
ELSE
	GrabPart_ON := FALSE;
END_IF
END_METHOD

PROPERTY PUBLIC GripperInPos0 : BOOL
GET
GripperInPos0 := NOT statPickPlaceInPositionCAxis90;
END_GET
END_PROPERTY

PROPERTY PUBLIC GripperInPos90 : BOOL
GET
GripperInPos90 := statPickPlaceInPositionCAxis90;
END_GET
END_PROPERTY

PROPERTY PUBLIC InPositionX_Y_Axis : BOOL
GET
InPositionX_Y_Axis := statPickPlaceInPositionXAxis AND statPickPlaceInPositionYAxis;
END_GET
END_PROPERTY

PROPERTY PUBLIC InPositionZAxis : BOOL
GET
InPositionZAxis := statPickPlaceInPositionZAxis;
END_GET
END_PROPERTY

METHOD PUBLIC MoveXYAxis_On : BOOL
VAR_INPUT
	StartMovePickPlaceX_YAxis	:	BOOL;
	Positions	:	PickPlacePosition;
END_VAR
IF OperatingMode.AutomaticIsActive AND OperatingMode.AutomaticStart.IsActive AND
	NOT statMovePickPlace AND StartMovePickPlaceX_YAxis
THEN
	IF (
    (Positions.PositionXAxis > statCurrentPositionXAxis + 0.1) OR
       (Positions.PositionXAxis < statCurrentPositionXAxis - 0.1) OR
       (Positions.PositionYAxis > statCurrentPositionYAxis + 0.1) OR
       (Positions.PositionYAxis < statCurrentPositionYAxis - 0.1)
	)  THEN
		SetPointXAxis := Positions.PositionXAxis;
		SetPointYAxis := Positions.PositionYAxis;
		statMovePickPlace := TRUE;
		statPickPlaceNewOrder := TRUE;
		MoveXYAxis_On := TRUE;
	ELSE		
		MoveXYAxis_On := FALSE;
	END_IF
ELSE
	MoveXYAxis_On := FALSE;
END_IF
END_METHOD

METHOD PUBLIC MoveZAxis_On : BOOL
VAR_INPUT
	StartMovePickPlaceZAxis	:	BOOL;
	Positions	:	PickPlacePosition;
END_VAR
IF OperatingMode.AutomaticIsActive AND OperatingMode.AutomaticStart.IsActive AND
	NOT statMovePickPlace AND StartMovePickPlaceZAxis THEN
	IF (Positions.PositionZAxis > statCurrentPositionZAxis + 0.1) OR
       (Positions.PositionZAxis < statCurrentPositionZAxis - 0.1) THEN
		SetPointZAxis := Positions.PositionZAxis;
		statMovePickPlace := TRUE;
		statPickPlaceNewOrder := TRUE;
		MoveZAxis_On := TRUE;
	ELSE
		MoveZAxis_On := FALSE;		
	END_IF
ELSE
	MoveZAxis_On := FALSE;
END_IF
END_METHOD

PROPERTY PUBLIC NewOrderActive : BOOL
GET
NewOrderActive := statPickPlaceNewOrder;
END_GET
END_PROPERTY

METHOD PUBLIC ReleasePart : BOOL
VAR_INPUT
	StartGrabPart	:	BOOL;
END_VAR
IF OperatingMode.AutomaticIsActive AND OperatingMode.AutomaticStart.IsActive AND
	InPositionX_Y_Axis AND InPositionZAxis AND StartGrabPart AND NOT statMovePickPlace 
THEN
	statGrabPart := FALSE;
	ReleasePart := TRUE;
ELSE
	ReleasePart := FALSE;
END_IF
END_METHOD

METHOD PUBLIC RotateGripperTo0 : BOOL
VAR_INPUT
	StartMovingGripperTo0	:	BOOL;
END_VAR
IF OperatingMode.AutomaticIsActive AND OperatingMode.AutomaticStart.IsActive AND
	InPositionX_Y_Axis AND InPositionZAxis AND StartMovingGripperTo0 AND NOT statMovePickPlace 
THEN
	statCAxisToPos90 := FALSE;
	RotateGripperTo0 := TRUE;
ELSE
	RotateGripperTo0 := FALSE;
END_IF
END_METHOD

METHOD PUBLIC RotateGripperTo90 : BOOL
VAR_INPUT
	StartMovingGripperTo90	:	BOOL;
END_VAR
IF OperatingMode.AutomaticIsActive AND OperatingMode.AutomaticStart.IsActive AND
	InPositionX_Y_Axis AND InPositionZAxis AND StartMovingGripperTo90 AND NOT statMovePickPlace 
THEN
	statCAxisToPos90 := TRUE;
	RotateGripperTo90 := TRUE;
ELSE
	RotateGripperTo90 := FALSE;
END_IF
END_METHOD

PROPERTY PUBLIC SetPointXAxis : REAL
GET
SetPointXAxis := statSetPointXAxis;
END_GET
SET
IF SetPointXAxis < 10.5 THEN
	statSetPointXAxis := SetPointXAxis;
END_IF
END_SET
END_PROPERTY

PROPERTY PUBLIC SetPointYAxis : Real
GET
END_GET
SET
IF SetPointYAxis < 1.25 THEN
	statSetPointYAxis := SetPointYAxis;	
END_IF
END_SET
END_PROPERTY

PROPERTY PUBLIC SetPointZAxis : REAL
GET
SetPointZAxis := statSetPointZAxis;
END_GET
SET
IF SetPointZAxis < 6.125 THEN
	statSetPointZAxis := SetPointZAxis;	
END_IF
END_SET
END_PROPERTY

END_FUNCTION_BLOCK

// ---- POUs/Vorlagen/PositingBar/FB_PositingBar.TcPOU
FUNCTION_BLOCK FB_PositingBar
VAR_INPUT
	PartIsClamped	:	BOOL;	//Positining bar is clamped
	VerticalLimitReached	:	BOOL;	//Positining bar Raised
	AlignmentDirection	:	PositingBarAlignmentDirection;	//Alingment of the positining bar
	ActorInstanceIndex	:	INT;	//Index in DropDown HMI
	ActorInstanceName	:	STRING;		//Name of the instance
END_VAR
VAR_OUTPUT
	Clamp	:	BOOL;	//1 = Positining bar should clamp, 0 = Positining bar should unclamp
	Raise	:	BOOL;	//1 = Positining bar should raise, 0 = Positining bar should lower
END_VAR
VAR_IN_OUT
	OperatingMode	:	OperatingMode;	//Schnittstelle für Betriebsarten
	HMIInterface	:	MachineSectionHMIInterface;	//HMI-Interface
END_VAR
VAR
	statExecuteClamp	:	BOOL;	//Internal command that the positining bar should clamp
	statExecuteRaise	:	BOOL;	//Internal command that the positining bar should raise
	statPositingBarIsClamped	:	BOOL;	//Internal feedback that positing bar is clamped (Property: IsClamped)
	statPositingBarIsRaised	:	BOOL;	//Internal feedback that positing bar is raised (Property: IsRaised)
	
	internOperatingMode	:	OperatingMode;	//Internal structure
	internHMIInterface	:	MachineSectionHMIInterface;	//Internal structure
	internInstanceActivatedFirstTime	:	BOOL;	//Instance the first time active
	internRisingEdgePressButtonClamp	:	R_TRIG;
	internRisingEdgePressButtonUnclamp	:	R_TRIG;
	internRisingEdgePressButtonRaise	:	R_TRIG;
	internRisingEdgePressButtonLower	:	R_TRIG;
END_VAR

(*===================== Operating Mode =====================*)
internOperatingMode := OperatingMode;
(*===================== HMI INTERFACE =====================*)
internHMIInterface := HMIInterface;

IF internHMIInterface.ActiveMachineSection = MachineSection.PositingBar AND
	internHMIInterface.SelectedActor = ActorInstanceIndex THEN
	(*===================== Initializing HMI-Interface =====================*)
	IF NOT internInstanceActivatedFirstTime THEN
		FC_InitializingSettingLines(HMIInterface := internHMIInterface);
		internInstanceActivatedFirstTime := TRUE;
	END_IF
	(*===================== Button Handling Movement =====================*)
	internHMIInterface.Movements.MovementSettingLines[1].CaptionSettingLine := CONCAT('Positining bar horizontal ', ActorInstanceName);
	internHMIInterface.Movements.MovementSettingLines[1].VisibilitySettingLine := TRUE;
	
	internHMIInterface.Movements.MovementSettingLines[1].SettingLineButtons[1].IsVisibleButton := TRUE;
	internHMIInterface.Movements.MovementSettingLines[1].SettingLineButtons[1].IsVisibleAxisPosition := FALSE;
	internHMIInterface.Movements.MovementSettingLines[1].SettingLineButtons[1].IsEnabled := OperatingMode.ManuelIsActive AND NOT
									 														OperatingMode.EStop.IsActive AND NOT
																							OperatingMode.Fault.IsActive AND NOT
																							statPositingBarIsClamped;
	internHMIInterface.Movements.MovementSettingLines[1].SettingLineButtons[1].InPosition := statPositingBarIsClamped;
	internHMIInterface.Movements.MovementSettingLines[1].SettingLineButtons[1].CaptionButton := 'Clamp';
	internHMIInterface.Movements.MovementSettingLines[1].SettingLineButtons[1].PathImageButton := 'Images\Clamp.svg';
	
	internHMIInterface.Movements.MovementSettingLines[1].SettingLineButtons[3].IsVisibleButton := TRUE;
	internHMIInterface.Movements.MovementSettingLines[1].SettingLineButtons[3].IsVisibleAxisPosition := FALSE;
	internHMIInterface.Movements.MovementSettingLines[1].SettingLineButtons[3].IsEnabled := OperatingMode.ManuelIsActive AND NOT
									 														OperatingMode.EStop.IsActive AND NOT
																							OperatingMode.Fault.IsActive AND
																							statPositingBarIsClamped;
	internHMIInterface.Movements.MovementSettingLines[1].SettingLineButtons[3].InPosition := NOT statPositingBarIsClamped;
	internHMIInterface.Movements.MovementSettingLines[1].SettingLineButtons[3].CaptionButton := 'Unclamp';
	internHMIInterface.Movements.MovementSettingLines[1].SettingLineButtons[3].PathImageButton := 'Images\Unclamp.svg';
	
	internHMIInterface.Movements.MovementSettingLines[2].CaptionSettingLine := CONCAT('Positining bar vertical ', ActorInstanceName);
	internHMIInterface.Movements.MovementSettingLines[2].VisibilitySettingLine := TRUE;
	
	internHMIInterface.Movements.MovementSettingLines[2].SettingLineButtons[1].IsVisibleButton := TRUE;
	internHMIInterface.Movements.MovementSettingLines[2].SettingLineButtons[1].IsVisibleAxisPosition := FALSE;
	internHMIInterface.Movements.MovementSettingLines[2].SettingLineButtons[1].IsEnabled := OperatingMode.ManuelIsActive AND NOT
									 														OperatingMode.EStop.IsActive AND NOT
																							OperatingMode.Fault.IsActive AND NOT
																							statPositingBarIsRaised;
	internHMIInterface.Movements.MovementSettingLines[2].SettingLineButtons[1].InPosition := VerticalLimitReached AND statExecuteRaise;
	internHMIInterface.Movements.MovementSettingLines[2].SettingLineButtons[1].CaptionButton := 'Raise';
	internHMIInterface.Movements.MovementSettingLines[2].SettingLineButtons[1].PathImageButton := 'Images\UpElevator.svg';
	
	internHMIInterface.Movements.MovementSettingLines[2].SettingLineButtons[3].IsVisibleButton := TRUE;
	internHMIInterface.Movements.MovementSettingLines[2].SettingLineButtons[3].IsVisibleAxisPosition := FALSE;
	internHMIInterface.Movements.MovementSettingLines[2].SettingLineButtons[3].IsEnabled := OperatingMode.ManuelIsActive AND NOT
									 														OperatingMode.EStop.IsActive AND NOT
																							OperatingMode.Fault.IsActive AND
																							statPositingBarIsRaised;
	internHMIInterface.Movements.MovementSettingLines[2].SettingLineButtons[3].InPosition := VerticalLimitReached AND NOT statExecuteRaise;
	internHMIInterface.Movements.MovementSettingLines[2].SettingLineButtons[3].CaptionButton := 'Lower';
	internHMIInterface.Movements.MovementSettingLines[2].SettingLineButtons[3].PathImageButton := 'Images\DownElevator.svg';
	
	(*===================== Clamp =====================*)
	internRisingEdgePressButtonClamp(CLK := internHMIInterface.Movements.MovementSettingLines[1].SettingLineButtons[1].IsPressed);
	IF internRisingEdgePressButtonClamp.Q THEN
		statExecuteClamp := TRUE;
	END_IF
	(*===================== Unclamp =====================*)
	internRisingEdgePressButtonUnclamp(CLK := internHMIInterface.Movements.MovementSettingLines[1].SettingLineButtons[3].IsPressed);
	IF internRisingEdgePressButtonUnclamp.Q THEN
		statExecuteClamp := FALSE;
	END_IF
	(*===================== Raise =====================*)
	internRisingEdgePressButtonRaise(CLK := internHMIInterface.Movements.MovementSettingLines[2].SettingLineButtons[1].IsPressed);
	IF internRisingEdgePressButtonRaise.Q THEN
		statExecuteRaise := TRUE;
	END_IF
	(*===================== Lower =====================*)
	internRisingEdgePressButtonLower(CLK := internHMIInterface.Movements.MovementSettingLines[2].SettingLineButtons[3].IsPressed);
	IF internRisingEdgePressButtonLower.Q THEN
		statExecuteRaise := FALSE;
	END_IF
	
	(*===================== Write Interface =====================*)
	HMIInterface := internHMIInterface;
ELSE
		internInstanceActivatedFirstTime := FALSE;
END_IF

(*===================== Operating Mode =====================*)
statPositingBarIsClamped := PartIsClamped;
statPositingBarIsRaised := VerticalLimitReached AND statExecuteRaise;

(*===================== Outputs =====================*)
Clamp := statExecuteClamp;
Raise := statExecuteRaise;
OperatingMode.Fault := internOperatingMode.Fault;

PROPERTY PUBLIC IsClamped : BOOL
GET
IsClamped := statPositingBarIsClamped;
END_GET
END_PROPERTY

PROPERTY PUBLIC LimitVerticalReached : BOOL
GET
LimitVerticalReached := statPositingBarIsRaised;
END_GET
END_PROPERTY

METHOD PUBLIC PositingBarClamping : BOOL
VAR_INPUT
	ClampPositiningBar	:	BOOL;
END_VAR
IF internOperatingMode.AutomaticIsActive AND internOperatingMode.AutomaticStart.IsActive AND NOT
	internOperatingMode.Fault.IsActive AND NOT internOperatingMode.EStop.IsActive AND NOT
	IsClamped AND ClampPositiningBar THEN
	statExecuteClamp := TRUE;
	PositingBarClamping := TRUE;
ELSE
	PositingBarClamping := FALSE;		
END_IF
END_METHOD

METHOD PUBLIC PositingBarLower : BOOL
VAR_INPUT
	LowerPositiningBar	:	BOOL;
END_VAR
IF internOperatingMode.AutomaticIsActive AND internOperatingMode.AutomaticStart.IsActive AND NOT
	internOperatingMode.Fault.IsActive AND NOT internOperatingMode.EStop.IsActive AND 
	LowerPositiningBar THEN
	statExecuteRaise := FALSE;
	PositingBarLower := TRUE;
ELSE
	PositingBarLower := FALSE;		
END_IF
END_METHOD

METHOD PUBLIC PositingBarRaise : BOOL
VAR_INPUT
	RaisePositiningBar	:	BOOL;
END_VAR
IF internOperatingMode.AutomaticIsActive AND internOperatingMode.AutomaticStart.IsActive AND NOT
	internOperatingMode.Fault.IsActive AND NOT internOperatingMode.EStop.IsActive AND
	RaisePositiningBar
THEN
	statExecuteRaise := TRUE;
	PositingBarRaise := TRUE;
ELSE
	PositingBarRaise := FALSE;		
END_IF
END_METHOD

METHOD PUBLIC PositingBarUnclamping : BOOL
VAR_INPUT
	UnclampPositiningBar	:	BOOL;
END_VAR
IF internOperatingMode.AutomaticIsActive AND internOperatingMode.AutomaticStart.IsActive AND NOT
	internOperatingMode.Fault.IsActive AND NOT internOperatingMode.EStop.IsActive AND 
	UnclampPositiningBar THEN
	statExecuteClamp := FALSE;
	PositingBarUnclamping := TRUE;
ELSE
	PositingBarUnclamping := FALSE;		
END_IF
END_METHOD

END_FUNCTION_BLOCK

// ---- POUs/Vorlagen/Remover/FB_Remover.TcPOU
FUNCTION_BLOCK FB_Remover
VAR_INPUT
	PartPresent	:	BOOL;
	ActorInstanceIndex	:	INT;
	ActorInstanceName	:	STRING;
END_VAR
VAR_IN_OUT
	HMIInterface	:	MachineSectionHMIInterface;
END_VAR
VAR_OUTPUT
	RemovePart	:	BOOL;
END_VAR
VAR
	internRemovePart	: BOOL;
	
	internHMIInterface	:	MachineSectionHMIInterface;
	internInstanceActivatedFirstTime	:	BOOL;
	internRisingEdgePressButton	:	R_TRIG;
END_VAR

(*===================== HMI Interface =====================*)
internHMIInterface := HMIInterface;

IF internHMIInterface.ActiveMachineSection = MachineSection.Remover AND
	internHMIInterface.SelectedActor = ActorInstanceIndex THEN
	(*===================== Initializing HMI-Interface =====================*)
	IF NOT internInstanceActivatedFirstTime THEN
		FC_InitializingSettingLines(HMIInterface := internHMIInterface);
		internInstanceActivatedFirstTime := TRUE;
	END_IF
	(*===================== Button Handling =====================*)
	internHMIInterface.Workpiece.WorkpieceSettingLines[1].CaptionSettingLine := CONCAT('Removing Part ', ActorInstanceName);
	internHMIInterface.Workpiece.WorkpieceSettingLines[1].VisibilitySettingLine := TRUE;
	
	internHMIInterface.Workpiece.WorkpieceSettingLines[1].SettingLineButtons[1].IsVisibleButton := TRUE;
	internHMIInterface.Workpiece.WorkpieceSettingLines[1].SettingLineButtons[1].IsVisibleAxisPosition := FALSE;
	internHMIInterface.Workpiece.WorkpieceSettingLines[1].SettingLineButtons[1].IsEnabled := NOT PartPresent;
	internHMIInterface.Workpiece.WorkpieceSettingLines[1].SettingLineButtons[1].InPosition := PartPresent;
	internHMIInterface.Workpiece.WorkpieceSettingLines[1].SettingLineButtons[1].CaptionButton := 'Remove';
	internHMIInterface.Workpiece.WorkpieceSettingLines[1].SettingLineButtons[1].PathImageButton := 'Images\RemovePartRemover.svg';
	
	internRisingEdgePressButton(CLK := internHMIInterface.Workpiece.WorkpieceSettingLines[1].SettingLineButtons[1].IsPressed);
	IF internRisingEdgePressButton.Q THEN
		internRemovePart := TRUE;
	END_IF
	(*===================== Write Interface =====================*)
	HMIInterface := internHMIInterface;
ELSE
		internInstanceActivatedFirstTime := FALSE;
END_IF
(*===================== Remove Parts =====================*)

IF NOT PartPresent THEN
	internRemovePart := FALSE;
END_IF

RemovePart := internRemovePart;

METHOD PUBLIC Remove : BOOL
IF PartPresent THEN
	internRemovePart := TRUE;
	Remove := TRUE;
ELSE
	internRemovePart := FALSE;
	Remove := FALSE;
END_IF
END_METHOD

END_FUNCTION_BLOCK

